	cfg.lrThld_Prevac := 5.0;	// Prevacuum pressure threshold
	// Cryo pressure threshold to start Turbo Pump before opening Valve
	cfg.lrThld_TP_SafeStartPressure := 0.01;	
	// Cryo pressure threshold to start Turbo Pump once Valve is open
	cfg.lrThld_Valve_SafeOpenPressure := 0.1;	
	cfg.tDelay := T#3S;	// Time delay before stopping Turbo Pump

	stat.bConfigured	:= TRUE;;
ELSE
	RETURN;	// Nothing to do any more
END_IF
END_METHOD

METHOD M_ExecuteControllers
VAR_INPUT
END_VAR
//
// Specific Cryo Lab Evacuation System HW configuration.
//

// Roughing Pump	
rp(	
	in_bSimulation	:= FALSE,
	in_sName		:= 'ECODRY V01',
	in_bEnable		:= ctrl.bEnable_RP,
	in_nSlaveID		:= 31,
	in_sVersion		:= 'V01',
	in_nPeriod		:= 2000);

// Turbo Molecular Pump
tp(	
	in_bSimulation	:= FALSE,
	in_sName		:= 'ATH2303M',
	in_bEnable		:= ctrl.bEnable_TP,
	in_nModel		:= 2303,
	in_bAutoMonitor	:= TRUE,
	in_nPeriod		:= 2000);

// Valve
valve(
	in_bEnable		:= ctrl.bEnable_Valve,
	in_nFeedback	:= E_CRYO_BIN_ACT_FEEDBACK.ON_AND_OFF);
END_METHOD

END_FUNCTION_BLOCK

// POUs/Subsystems/Examples/Evacuation/FB_CRYO_EVAC_PDS
FUNCTION_BLOCK FB_CRYO_EVAC_PDS EXTENDS FB_CRYO_EVAC_BASE
VAR_INPUT
END_VAR
VAR_OUTPUT
END_VAR
VAR
	rp:	FB_CRYO_PUMP_MVP030;	// Roughing Pump
	tp:	FB_CRYO_PUMP_HIPACE30;	// Turbo Molecular Pump
	
END_VAR

SUPER^();

METHOD M_Configure
VAR_INPUT
END_VAR
//
// Specific PDS IR Imager configuration.
//
IF NOT stat.bConfigured	THEN
	// MANDATORY: Set References !!!
	// If not done, system will crash !!!
	rpRef	REF=rp;
	tpRef	REF=tp;
	

	// Specific instance configuration, e.g. anything different
	// from the default values given in the cfg structure of type T_CRYO_EVAC_CFG.
	cfg.nPressGaugeType1	:= E_CRYO_SENSOR_TYPE_PRESS.PKR_360;
	cfg.nPressGaugeType2	:= E_CRYO_SENSOR_TYPE_PRESS.PKR_360;

	cfg.lrThld_Prevac := 5.0;	// Prevacuum pressure threshold
	// Cryo pressure threshold to start Turbo Pump before opening Valve
	cfg.lrThld_TP_SafeStartPressure := 0.01;	
	// Cryo pressure threshold to start Turbo Pump once Valve is open
	cfg.lrThld_Valve_SafeOpenPressure := 0.1;	
	
	cfg.tDelay := T#3S;	// Time delay before stopping Turbo Pump

	stat.bConfigured	:= TRUE;;
ELSE
	RETURN;	// Nothing to do any more
END_IF
END_METHOD

METHOD M_ExecuteControllers
VAR_INPUT
END_VAR
//
// Specific PDS IR Imager HW.
//

// Roughing Pump	
rp(	
	in_bSimulation	:= FALSE,
	in_sName		:= 'MVP 030',
	in_bEnable		:= ctrl.bEnable_RP,
	in_nModel		:= 30,
	in_bAutoMonitor	:= TRUE,
	in_nPeriod		:= 3000);

// Turbo Molecular Pump
tp(	
	in_bSimulation	:= FALSE,
	in_sName		:= 'HIPACE 30',
	in_bEnable		:= ctrl.bEnable_TP,
	in_nModel		:= 30,
	in_bAutoMonitor	:= TRUE,
	in_nPeriod		:= 3000);


valve(in_bEnable	:= ctrl.bEnable_Valve);
END_METHOD

END_FUNCTION_BLOCK

// POUs/Subsystems/Examples/Evacuation/FB_SIM_MICADO_PUMPS
FUNCTION_BLOCK FB_SIM_MICADO_PUMPS
VAR_INPUT
	in_RefPVP:	REFERENCE TO FB_CRYO_PUMP_ECODRY;
	in_RefTMP:	REFERENCE TO FB_CRYO_PUMP_ATH2303M;
	in_Delay:	TIME := T#10S;
END_VAR
VAR_OUTPUT
END_VAR
VAR
	trgStart_PVP:	R_TRIG;
	trgStart_TMP:	R_TRIG;
	trgStop_PVP:	F_TRIG;
	trgStop_TMP:	F_TRIG;
	
	timer_PVP:		TON;
	timer_TMP:		TON;
	
	bON_PVP:		BOOL := FALSE;
	bON_TMP:		BOOL := FALSE;
	
	q_PVP_Running	AT %Q*:	BOOL := TRUE;	// Active low!
	q_TMP_Ready		AT %Q*:	BOOL;
	q_TMP_Speed100	AT %Q*:	BOOL;
	
	ptrTMP_Speed:	POINTER TO DINT;
END_VAR

// Assign pointer to TMP speed.
ptrTMP_Speed	:= ADR(in_RefTMP.stat.nPumpSpeed);

// Get Start signals
trgStart_PVP(CLK:=in_RefPVP.in_bEnable);
trgStart_TMP(CLK:=in_RefTMP.in_bEnable);

// Get Stop signals
trgStop_PVP(CLK:=in_RefPVP.in_bEnable);
trgStop_TMP(CLK:=in_RefTMP.in_bEnable);

// Start timer on Start/Stop events
IF trgStart_PVP.Q THEN
	bON_PVP	:= TRUE;
	timer_PVP(IN:=FALSE);
	timer_PVP(IN:=TRUE, PT:=in_Delay/2);
ELSIF trgStop_PVP.Q THEN
	bON_PVP	:= FALSE;
	timer_PVP(IN:=FALSE);
	timer_PVP(IN:=TRUE, PT:=in_Delay/2);
END_IF

IF trgStart_TMP.Q THEN
	bON_TMP	:= TRUE;
	timer_TMP(IN:=FALSE);
	timer_TMP(IN:=TRUE, PT:=in_Delay);
ELSIF trgStop_TMP.Q THEN
	bON_TMP	:= FALSE;
	timer_TMP(IN:=FALSE);
	timer_TMP(IN:=TRUE, PT:=in_Delay * 2);
END_IF

// Execute timers
timer_PVP();
timer_TMP();

// Set outputs on timer expiry
IF timer_PVP.Q THEN
	// NOTE: PVP feedback is active low.
	IF bON_PVP THEN
		q_PVP_Running	:= FALSE;
	ELSE
		q_PVP_Running	:= TRUE;
	END_IF
END_IF

IF bON_TMP  AND (NOT timer_TMP.Q AND timer_TMP.ET > T#3S) THEN
	// Starting up.
	// Set speed > 100 rpm after 3 sec.
	ptrTMP_Speed^	:= 500;
	q_TMP_Speed100	:= TRUE;
END_IF

IF NOT bON_TMP  AND (NOT timer_TMP.Q AND timer_TMP.ET > T#5S) THEN
	// Stopping the pump.
	// Not ready after 5 sec.
	// However, the pump is still spinning.
	ptrTMP_Speed^	:= 1800;
	q_TMP_Ready		:= FALSE;
END_IF

IF timer_TMP.Q THEN
	IF bON_TMP THEN
		ptrTMP_Speed^	:= 2000;
		q_TMP_Ready	:= TRUE;
	ELSE
		ptrTMP_Speed^	:= 0;
		q_TMP_Ready		:= FALSE;
		q_TMP_Speed100	:= FALSE;
	END_IF
END_IF

END_FUNCTION_BLOCK

// POUs/Subsystems/Examples/Evacuation/FB_SIM_MICADO_VALVES
FUNCTION_BLOCK FB_SIM_MICADO_VALVES
VAR_INPUT
END_VAR
VAR_OUTPUT
END_VAR
VAR
	// Output valve control signals
	i_bON_PVV1	AT %I*:	BOOL;
	i_bON_PVV2	AT %I*:	BOOL;
	i_bON_PVV3	AT %I*:	BOOL;
	i_bON_PVV4	AT %I*:	BOOL;
	i_bON_GBV	AT %I*:	BOOL;
	
	
	// Simulation of ON/open feedback signal
	q_bON_PVV1	AT %Q*:	BOOL := FALSE;
	q_bON_PVV2	AT %Q*:	BOOL := FALSE;
	q_bON_PVV3	AT %Q*:	BOOL := FALSE;
	q_bON_PVV4	AT %Q*:	BOOL := FALSE;
	q_bON_GBV	AT %Q*:	BOOL := FALSE;
	
	// Simulation of OFF/closed feedback signal
	q_bOFF_PVV1	AT %Q*:	BOOL := TRUE;
	q_bOFF_PVV2	AT %Q*:	BOOL := TRUE;
	q_bOFF_PVV3	AT %Q*:	BOOL := TRUE;
	q_bOFF_PVV4	AT %Q*:	BOOL := TRUE;
	q_bOFF_GBV	AT %Q*:	BOOL := TRUE;
	

END_VAR

// ON signals are active low
q_bON_PVV1	:= i_bON_PVV1;
q_bON_PVV2	:= i_bON_PVV2;
q_bON_PVV3	:= i_bON_PVV3;
q_bON_PVV4	:= i_bON_PVV4;
q_bON_GBV	:= i_bON_GBV;


// OFF signals are active low
q_bOFF_PVV1	:= NOT i_bON_PVV1;
q_bOFF_PVV2	:= NOT i_bON_PVV2;
q_bOFF_PVV3	:= NOT i_bON_PVV3;
q_bOFF_PVV4	:= NOT i_bON_PVV4;
q_bOFF_GBV	:= NOT i_bON_GBV;

END_FUNCTION_BLOCK

// POUs/Subsystems/Examples/LN2_Precooling/FB_CRYO_LN2_PRECOOL
FUNCTION_BLOCK FB_CRYO_LN2_PRECOOL EXTENDS FB_CRYO_GEN_CTRL_BASE
VAR_INPUT
	in_lrTempK:				LREAL;			// Temperature input value [K]
	in_bTempValid:			BOOL := TRUE;	// Temperature Valid flag
	// Two parameters for decision making
	in_lrTempValveOpen:		LREAL := 91.27;		// Open  valve if temperature above this value [K]
	in_lrTempValveClose:	LREAL := 79.148;	// Close valve if temperature below this value [K]
END_VAR
VAR_OUTPUT
END_VAR
VAR
	// Status structure
	{attribute 'OPC.UA.DA' := '1'}
	stat:				T_CRYO_GEN_CTRL_STATUS_BASE;
	
	// LN2 valve
	valve:				FB_CRYO_VALVE_CTRL;
	bEnable_valve:		BOOL := FALSE;	// Valve open when bEnable_valve = TRUE
		

END_VAR

SUPER^();

METHOD M_ActionOffExecute
VAR_INPUT
END_VAR
//
// In this method the Enable flag of the valve is set to FALSE,
// meaning close the valve.
// 
// In the corresponding Activity M_ActivitySwitchingOff(), 
// the completion of the CLOSE/OFF command will be checked.
//
timer(IN:=FALSE);	// Reset Timer - mandatory!

// Close the valve
bEnable_valve	:= FALSE;
END_METHOD

METHOD M_ActionOnExecute
VAR_INPUT
END_VAR
//
// In this method the Enable flag of the valve is set to TRUE,
// meaning open the valve.
// 
// In the corresponding Activity M_ActivitySwitchingOn(), 
// the completion of the OPEN/ON command will be checked.
//
timer(IN:=FALSE);	// Reset Timer - mandatory!

// Close the valve
bEnable_valve	:= TRUE;
END_METHOD

METHOD M_ActivitySwitchingOff : BOOL
VAR_INPUT
END_VAR
//
// Wait for the valve to CLOSE/OFF.
// The valve state is available in its status structure.
// When complete, the method shall return TRUE, otherwise FALSE.


//
// Execute the timer - mandatory.
// Timer expiry is checked in M_ProcessEvents().
//
timer(IN:=TRUE, PT:=UDINT_TO_TIME(in_nTimeout));
	
// If valve is closed, return TRUE, otherwise FALSE.
IF valve.stat.bActOFF THEN
	M_ActivitySwitchingOff := TRUE;
ELSE
	M_ActivitySwitchingOff := FALSE;
END_IF
END_METHOD

METHOD M_ActivitySwitchingOn : BOOL
VAR_INPUT
END_VAR
//
// Wait for the valve to OPEN/ON.
// The valve state is available in its status structure.
// When complete, the method shall return TRUE, otherwise FALSE.


//
// Execute the timer - mandatory.
// Timer expiry is checked in M_ProcessEvents().
//
timer(IN:=TRUE, PT:=UDINT_TO_TIME(in_nTimeout));
	
// If valve is open, return TRUE, otherwise FALSE.
IF valve.stat.bActON THEN
	M_ActivitySwitchingOn := TRUE;
ELSE
	M_ActivitySwitchingOn := FALSE;
END_IF
END_METHOD

METHOD M_Configure
VAR_INPUT
END_VAR
// Configure the system and set the bConfigured flag to TRUE.

(*
	TODO USER: 
	- Set references to extended structures. e.g.
	     statRef REF=stat;
	- Configure the system.
*)

//	MUST be the very first line!!!
statRef REF=stat;

// The system has been configured
bConfigured := TRUE;
END_METHOD

METHOD M_ControlLoop : BOOL
VAR_INPUT
END_VAR
//
// This method implements the logic for controlling the LN2 valve.
// 
// The return value indicates if the valve should be OPEN/TRUE or CLOSED/FALSE
//
	
CASE statRef.nState OF
	E_CRYO_BIN_CTRL_STATE.ACTIVE_SWITCHING_ON,
	E_CRYO_BIN_CTRL_STATE.ACTIVE_ON:
		IF in_bTempValid AND in_lrTempK < in_lrTempValveClose THEN
			// Temperature too low.
			// Close the valve to stop cooling.
			M_ControlLoop	:= FALSE;
		ELSE
			// Keep the valve open
			M_ControlLoop	:= TRUE;
		END_IF

	E_CRYO_BIN_CTRL_STATE.ACTIVE_SWITCHING_OFF,
	E_CRYO_BIN_CTRL_STATE.ACTIVE_OFF:
		IF in_bTempValid AND in_lrTempK > in_lrTempValveOpen THEN
			// Temperature too high.
			// Open the valve to start cooling.
			M_ControlLoop	:= TRUE;
		ELSE
			// Keep the valve closed
			M_ControlLoop	:= FALSE;
		END_IF
ELSE
	// Keep the valve closed
	M_ControlLoop	:= FALSE;
END_CASE
END_METHOD

METHOD M_ExecuteActuators
VAR_INPUT
END_VAR
(*
	TODO USER: Execute all actuators, e.g. valve, heater, etc.
*)

valve(	in_nTimeout	:= 3000, 
		in_bEnable	:= bEnable_valve);
END_METHOD

METHOD M_IsError : BOOL
VAR_INPUT
END_VAR
//
// Check all possible failure conditions.
//
// This includes:
// - Configuration,
// - Validity of temperature reading,
// - Valve failure.
// 
// Return TRUE in case of errors.
// Set error description as well.
//
IF in_lrTempValveClose >= in_lrTempValveOpen THEN
	// The temperatue at which valve opens must be
	// higher than the one at which it closes.
	M_IsError	:= TRUE;
	stat.sError	:= 'ERROR: Wrong temperature limits!';
ELSIF NOT in_bTempValid	THEN
	// Temperature reading invalid.
	M_IsError	:= TRUE;
	stat.sError	:= 'ERROR: Reference temperature invalid!';
ELSIF valve.stat.bError 	THEN
	// Valve has failed.
	M_IsError	:= TRUE;
	stat.sError	:= 'ERROR: Valve failure!';
ELSE
	M_IsError	:= FALSE;
END_IF
END_METHOD

METHOD M_SetStatus
VAR_INPUT
END_VAR
// Execute M_SetStatus() of the base FB
SUPER^.M_SetStatus();


// Correct for LN2 specific labels

CASE statRef.nState OF
	
	E_CRYO_BIN_CTRL_STATE.ACTIVE_OFF:
	statRef.sState	:= 'ACTIVE_VALVE_CLOSED';
	
	E_CRYO_BIN_CTRL_STATE.ACTIVE_ON:
	statRef.sState	:= 'ACTIVE_VALVE_OPEN';
	
	E_CRYO_BIN_CTRL_STATE.ACTIVE_SWITCHING_ON:
	statRef.sState	:= 'OPENING VALVE...';
	
	E_CRYO_BIN_CTRL_STATE.ACTIVE_SWITCHING_OFF:
	statRef.sState	:= 'CLOSING VALVE...';
	
END_CASE
END_METHOD

END_FUNCTION_BLOCK

// POUs/Subsystems/Examples/LN2_Precooling/FB_SIM_LN2_PRECOOL
FUNCTION_BLOCK FB_SIM_LN2_PRECOOL
VAR_INPUT
	ln2Ref:	REFERENCE TO FB_CRYO_LN2_PRECOOL;
END_VAR
VAR_OUTPUT
	lrTempK:	LREAL;	// Simulated temperature value [K]
END_VAR
VAR
	SIM_ln2_temp:	FB_CRYO_SIM_TEMPERATURE;	// Simulated temperature FB
	
	trgEnable:		R_TRIG;						// Precooling  enable change trigger
	trgDisable:		F_TRIG;						// Precooling disable change trigger
	trgState:		R_TRIG;						// State change trigger

	nState:			E_CRYO_BIN_CTRL_STATE	:= E_CRYO_BIN_CTRL_STATE.NONE;
	
END_VAR

// Detect change of LN2 system Enable 
trgEnable(CLK := ln2Ref.in_bEnable);

// Detect change of LN2 system Disable 
trgDisable(CLK := ln2Ref.in_bEnable);

// Detect change of LN2 system State 
trgState(CLK := (	(ln2Ref.stat.nState = E_CRYO_BIN_CTRL_STATE.ACTIVE_ON OR 
					 ln2Ref.stat.nState = E_CRYO_BIN_CTRL_STATE.ACTIVE_OFF) 	AND 
					ln2Ref.stat.nState <> nState));

IF trgEnable.Q	THEN
	// System enabled.

	// Save current state
	nState	:= ln2Ref.stat.nState;
	
	// Start changing temperature just to get the system 
	// working for the first time.
	IF SIM_ln2_temp.lrTempK >= ln2Ref.in_lrTempValveClose	THEN
		// Lower simulated temperature to lower limit -1 deg in 5 sec.
		SIM_ln2_temp.M_RampTo(ln2Ref.in_lrTempValveClose - 1, 5000);
	ELSE
		// Rise simulated temperature to upper limit +1 deg in 5 sec.
		SIM_ln2_temp.M_RampTo(ln2Ref.in_lrTempValveOpen + 1, 5000);
	END_IF
ELSIF trgDisable.Q	THEN
	// System disabled. Stop the temperature ramp.
	SIM_ln2_temp.M_Stop();	
ELSIF ln2Ref.in_bEnable AND trgState.Q	THEN
	// State of enabled system changed.
	// Save new state
	nState	:= ln2Ref.stat.nState;
	
	// Start a ramp, depending on the new state.
	IF ln2Ref.stat.nState = E_CRYO_BIN_CTRL_STATE.ACTIVE_ON	THEN
		// Valve open, the temperature should start falling.
		// Ramp it down to the CLOSE limit minus 1 deg in 10 sec.
		SIM_ln2_temp.M_RampTo(ln2Ref.in_lrTempValveClose - 1.0, 10000);
	ELSIF ln2Ref.stat.nState = E_CRYO_BIN_CTRL_STATE.ACTIVE_OFF	THEN
		// Valve closed, the temperature should start rising.
		// Ramp it up to the OPEN limit plus 1 deg in 10 sec.
		SIM_ln2_temp.M_RampTo(ln2Ref.in_lrTempValveOpen + 1.0, 10000);
	END_IF
END_IF


// Execute temperature simulator FB.
SIM_ln2_temp();

// Assign the simulated temperature to the output var
lrTempK	:= SIM_ln2_temp.lrTempK;

END_FUNCTION_BLOCK

// POUs/Utilities/FB_CRYO_THLD_BASE
FUNCTION_BLOCK FB_CRYO_THLD_BASE
VAR_INPUT
	in_nMode:		E_CRYO_THLD_MODE := E_CRYO_THLD_MODE.FIXED;
	in_aThld:		ARRAY [1..4] OF LREAL;	// Array of fixed thresholds. See E_CRYO_ALARM_LEVELS and E_CRYO_ALARM_IDX.
	in_aThldDelay:	ARRAY [1..4] OF UDINT;	// Array of delays for each threshold [ms].
	in_lrHyst:		LREAL := 0.0;			// Hysteresis value, percent or absolute (see in_bHystPct)
	in_bHystPct:	BOOL := TRUE;			// If TRUE, hysteresis is in %, otherwise absolute value.
	in_lrValue:		LREAL;					// Value to compare against the thresholds
	in_lrPar1:		LREAL := 0.0;			// Par1, e.g. temperature, for ACTIVE thresholds
END_VAR
VAR_OUTPUT
	out_aThld:			ARRAY [1..4] OF LREAL;	// Active thresholds
	out_nAlarmState:	E_CRYO_ALARM_LEVEL	:= E_CRYO_ALARM_LEVEL.NORMAL;	// Alarm state, e.g. ALARM_HIGH
	out_sAlarmState:	STRING := 'NORMAL';	// Alarm state as a string, e.g. 'ALARM HIGH'
END_VAR
VAR
	timer:	TON;
END_VAR

// Set thresholds
M_SetThresholds();

// Compare input value against the thresholds
M_CheckAlarms();

METHOD M_CheckAlarms : BOOL
VAR_INPUT
END_VAR
VAR
	lrHyst:	LREAL;
END_VAR

// Execute the delay timer.
timer();

//
// Check the input value against the thresholds
// and set alarms and warnings.
// If configured for, activate alarms after a delay.
// Note: the value is compared against the OUT Thresholds !!!
//
CASE out_nAlarmState OF
	E_CRYO_ALARM_LEVEL.NORMAL:
		IF in_lrValue > out_aThld[E_CRYO_ALARM_IDX.ALARM_HIGH] THEN
			IF in_aThldDelay[E_CRYO_ALARM_IDX.ALARM_HIGH] > 0	THEN
				// Activation delay is configured.
				// Start the timer and change state to WARNING_HIGH.
				timer(IN:=FALSE);
				timer(IN:=TRUE, PT:=UDINT_TO_TIME(in_aThldDelay[E_CRYO_ALARM_IDX.ALARM_HIGH]));
				out_nAlarmState	:= E_CRYO_ALARM_LEVEL.WARNING_HIGH;
			ELSE
				timer(IN:=FALSE);
				out_nAlarmState	:= E_CRYO_ALARM_LEVEL.ALARM_HIGH;
			END_IF
		ELSIF in_lrValue < out_aThld[E_CRYO_ALARM_IDX.ALARM_LOW] THEN
			IF in_aThldDelay[E_CRYO_ALARM_IDX.ALARM_LOW] > 0	THEN
				// Activation delay is configured.
				// Start the timer and change state to WARNING_LOW.
				timer(IN:=FALSE);
				timer(IN:=TRUE, PT:=UDINT_TO_TIME(in_aThldDelay[E_CRYO_ALARM_IDX.ALARM_LOW]));
				out_nAlarmState	:= E_CRYO_ALARM_LEVEL.WARNING_LOW;
			ELSE
				timer(IN:=FALSE);
				out_nAlarmState	:= E_CRYO_ALARM_LEVEL.ALARM_LOW;
			END_IF
		ELSIF in_lrValue > out_aThld[E_CRYO_ALARM_IDX.WARNING_HIGH] THEN
			IF in_aThldDelay[E_CRYO_ALARM_IDX.WARNING_HIGH] > 0	THEN
				// Activation delay is configured.
				// Activate the warning once the timer expires.
				timer(IN:=TRUE, PT:=UDINT_TO_TIME(in_aThldDelay[E_CRYO_ALARM_IDX.WARNING_HIGH]));
				IF timer.Q	THEN
					IF in_lrValue > out_aThld[E_CRYO_ALARM_IDX.ALARM_HIGH] THEN
						// It might be that due to the delay the alarm level has been reached.
						out_nAlarmState	:= E_CRYO_ALARM_LEVEL.ALARM_HIGH;
					ELSE
						out_nAlarmState	:= E_CRYO_ALARM_LEVEL.WARNING_HIGH;
					END_IF
				END_IF
			ELSE
				timer(IN:=FALSE);
				out_nAlarmState	:= E_CRYO_ALARM_LEVEL.WARNING_HIGH;
			END_IF
		ELSIF	in_lrValue < out_aThld[E_CRYO_ALARM_IDX.WARNING_LOW]	THEN
			IF in_aThldDelay[E_CRYO_ALARM_IDX.WARNING_LOW] > 0	THEN
				// Activation delay is configured.
				// Activate the warning once the timer expires.
				timer(IN:=TRUE, PT:=UDINT_TO_TIME(in_aThldDelay[E_CRYO_ALARM_IDX.WARNING_LOW]));
				IF timer.Q	THEN
					IF in_lrValue < out_aThld[E_CRYO_ALARM_IDX.ALARM_LOW] THEN
						// It might be that due to the delay the alarm level has been reached.
						out_nAlarmState	:= E_CRYO_ALARM_LEVEL.ALARM_LOW;
					ELSE
						out_nAlarmState	:= E_CRYO_ALARM_LEVEL.WARNING_LOW;
					END_IF
				END_IF
			ELSE
				timer(IN:=FALSE);
				out_nAlarmState	:= E_CRYO_ALARM_LEVEL.WARNING_LOW;
			END_IF
		ELSE
			timer(IN:=FALSE);
		END_IF
	E_CRYO_ALARM_LEVEL.WARNING_HIGH:
		lrHyst	:= M_GetHysteresis(E_CRYO_ALARM_IDX.WARNING_HIGH);
		IF	in_lrValue > out_aThld[E_CRYO_ALARM_IDX.ALARM_HIGH]	THEN
			IF in_aThldDelay[E_CRYO_ALARM_IDX.ALARM_HIGH] > 0	THEN
				// Activation delay is configured.
				// Activate the alarm once the timer expires.
				timer(IN:=TRUE, PT:=UDINT_TO_TIME(in_aThldDelay[E_CRYO_ALARM_IDX.ALARM_HIGH]));
				IF timer.Q	THEN
					out_nAlarmState	:= E_CRYO_ALARM_LEVEL.ALARM_HIGH;
				END_IF
			ELSE
				timer(IN:=FALSE);
				out_nAlarmState	:= E_CRYO_ALARM_LEVEL.ALARM_HIGH;
			END_IF
		ELSIF in_lrValue < (out_aThld[E_CRYO_ALARM_IDX.WARNING_HIGH] - lrHyst) THEN
			timer(IN:=FALSE);
			out_nAlarmState	:= E_CRYO_ALARM_LEVEL.NORMAL;
		ELSE
			timer(IN:=FALSE);
		END_IF
	E_CRYO_ALARM_LEVEL.WARNING_LOW:
		lrHyst	:= M_GetHysteresis(E_CRYO_ALARM_IDX.WARNING_LOW);
		IF	in_lrValue < out_aThld[E_CRYO_ALARM_IDX.ALARM_LOW]	THEN
			IF in_aThldDelay[E_CRYO_ALARM_IDX.ALARM_LOW] > 0	THEN
				// Activation delay is configured.
				// Activate the alarm once the timer expires.
				timer(IN:=TRUE, PT:=UDINT_TO_TIME(in_aThldDelay[E_CRYO_ALARM_IDX.ALARM_LOW]));
				IF timer.Q	THEN
					out_nAlarmState	:= E_CRYO_ALARM_LEVEL.ALARM_LOW;
				END_IF
			ELSE
				timer(IN:=FALSE);
				out_nAlarmState	:= E_CRYO_ALARM_LEVEL.ALARM_LOW;
			END_IF
		ELSIF in_lrValue > (out_aThld[E_CRYO_ALARM_IDX.WARNING_LOW] + lrHyst) THEN
			timer(IN:=FALSE);
			out_nAlarmState	:= E_CRYO_ALARM_LEVEL.NORMAL;
		ELSE
			timer(IN:=FALSE);
		END_IF
	E_CRYO_ALARM_LEVEL.ALARM_HIGH:
		lrHyst	:= M_GetHysteresis(E_CRYO_ALARM_IDX.ALARM_HIGH);
		IF in_lrValue < (out_aThld[E_CRYO_ALARM_IDX.ALARM_HIGH] - lrHyst) THEN
			out_nAlarmState	:= E_CRYO_ALARM_LEVEL.WARNING_HIGH;
		END_IF
	E_CRYO_ALARM_LEVEL.ALARM_LOW:
		lrHyst	:= M_GetHysteresis(E_CRYO_ALARM_IDX.ALARM_LOW);
		IF in_lrValue > (out_aThld[E_CRYO_ALARM_IDX.ALARM_LOW] + lrHyst) THEN
			out_nAlarmState	:= E_CRYO_ALARM_LEVEL.WARNING_LOW;
		END_IF
END_CASE

// Set alarm level labels
M_UserSetLabel(out_nAlarmState);
END_METHOD

METHOD M_GetHysteresis : LREAL
VAR_INPUT
	in_nIndex:	E_CRYO_ALARM_IDX;
END_VAR
VAR
	lrHyst:	LREAL;
END_VAR
//
// Get the absolute value of hysteresis.
// 
IF in_bHystPct THEN
	// The vaue is given as percentage of threshold.
	lrHyst	:= in_aThld[in_nIndex] * in_lrHyst / 100.0;
ELSE
	// The vaue is given as absolute value.
	lrHyst	:= in_lrHyst;
END_IF

M_GetHysteresis	:= ABS(lrHyst);
END_METHOD

METHOD M_SetThresholds : BOOL
VAR_INPUT
END_VAR
VAR
	i:	INT;
END_VAR
CASE in_nMode OF
	E_CRYO_THLD_MODE.FIXED:
		// Take the input array for thresholds
		FOR i:=1 TO 4 DO
			out_aThld[i]	:= in_aThld[i];
		END_FOR
	E_CRYO_THLD_MODE.ACTIVE:
		// Dynamically set thresholds
		M_UserSetActiveThresholds();
	E_CRYO_THLD_MODE.LAST_ACTIVE:
		// Keep last thresholds. Don't do anything.
		;
END_CASE
END_METHOD

METHOD M_UserSetActiveThresholds : BOOL
// This is a Dummy implementation of active thresholds.
// TODO User: Define specific implementation.
VAR_INPUT
END_VAR
VAR
	i:	INT;
END_VAR
// TODO User
// Define specific implementation.
// This is just an example.
//
out_aThld[E_CRYO_ALARM_IDX.ALARM_LOW]	:= in_aThld[E_CRYO_ALARM_IDX.ALARM_LOW]    + in_lrPar1;
out_aThld[E_CRYO_ALARM_IDX.WARNING_LOW]	:= in_aThld[E_CRYO_ALARM_IDX.WARNING_LOW]  + in_lrPar1;
out_aThld[E_CRYO_ALARM_IDX.WARNING_HIGH]	:= in_aThld[E_CRYO_ALARM_IDX.WARNING_HIGH] - in_lrPar1;
out_aThld[E_CRYO_ALARM_IDX.ALARM_HIGH]	:= in_aThld[E_CRYO_ALARM_IDX.ALARM_HIGH]   - in_lrPar1;
END_METHOD

METHOD M_UserSetLabel : BOOL
VAR_INPUT
	in_nLevel:	E_CRYO_ALARM_LEVEL;
END_VAR
//
// Set labels depending on the alarm level.
// This is the default implementation.
// To be overwritten by User if different labels are needed.
//
CASE in_nLevel OF
	E_CRYO_ALARM_LEVEL.ALARM_LOW:
		out_sAlarmState	:= 'ALARM LOW';
	E_CRYO_ALARM_LEVEL.WARNING_LOW:
		out_sAlarmState	:= 'WARNING LOW';
	E_CRYO_ALARM_LEVEL.NORMAL:
		out_sAlarmState	:= 'NORMAL';
	E_CRYO_ALARM_LEVEL.WARNING_HIGH:
		out_sAlarmState	:= 'WARNING HIGH';
	E_CRYO_ALARM_LEVEL.ALARM_HIGH:
		out_sAlarmState	:= 'ALARM HIGH';
END_CASE
END_METHOD

END_FUNCTION_BLOCK

// POUs/MAIN
PROGRAM MAIN
VAR
	
	
	{attribute 'OPC.UA.DA' := '1'}
	Cryo_Ctrl:	FB_CRYO_CTRL;
	
	
	{attribute 'OPC.UA.DA' := '1'}
	SIM_Cryo_Ctrl:	FB_CRYO_SIM_CTRL;
	
	//
	// Pressure voting system testing
	//
	P1_1:	FB_CRYO_SENSOR_PRESSURE;
	P1_2:	FB_CRYO_SENSOR_PRESSURE;
	P1_3:	FB_CRYO_SENSOR_PRESSURE;
	P1_4:	FB_CRYO_SENSOR_PRESSURE;
	P1_5:	FB_CRYO_SENSOR_PRESSURE;
	P1:		FB_CRYO_PRESSURE_VOTE;	// Voting of P1_1..P1_5

	nVoteMethod:		E_CRYO_VOTE	:=E_CRYO_VOTE.V_3oo5;
	bP1_Sim:			BOOL := FALSE;
	SIM_Pressure_P1:	FB_CRYO_SIM_PRESSURE;		// P1 Pressure simulator
	pressOR_P1:			FB_CRYO_CMD_OVERRIDE;

	////////////////////////////
	// Temperature testing
	//
	T1:		FB_CRYO_SENSOR_TEMPERATURE;
	T2:		FB_CRYO_TEMPERATURE;
	nRampPeriodSec:		UDINT := 60;	// Ramp measurement period [sec]. Default 60 sec.
	tempOR_T2:	FB_CRYO_CMD_OVERRIDE;
	simT2:		BOOL;
	////////////////////////////
	
	
	//////////////////////////////////////////////////////////////////
	
	//
	// Threshold testing
	//
	thld1:		FB_CRYO_THLD_BASE;	// Threshold handling
	
	// Threshold levels in format
	// [<alarm low>, <warning low>, <warning high>, <alarm high>]
	aThlds:		ARRAY [1..4] OF LREAL	:= [-80.0, -60.0, 40.0, 80.0];
	aThldDelay:	ARRAY [1..4] OF UDINT	:= [1000, 0, 2000, 0];
	nThldMode:	E_CRYO_THLD_MODE := E_CRYO_THLD_MODE.FIXED;	// Threshold check mode
	lrHyst:		LREAL	:= 10.0;	// Threshold hysteresis
	lrThldRef:	LREAL	:= 0.0;		// Threshold reference for User defined active thresholds
	
	SIM_thld1:	FB_CRYO_SIM_SINE;	// Simulated signal for threshold testing
	SIM_thld2:	FB_CRYO_SIM_SINE;	// Simulated signal for threshold testing
	nSimPer1:	UDINT := 60000;		// Period [ms] of simulated sine curve #1
	nSimPer2:	UDINT := 16000;		// Period [ms] of simulated sine curve #2
	
	/////////////////////////////////////////////////////////////////////////
	/////////////////////////////////////////////////////////////////////////

	///////////////////
	// Lakeshore 336
	///////////////////
	// Lakeshore 336 (Ethernet interface)
	{attribute 'OPC.UA.DA' := '1'}
	LS336_TCP:		FB_LAKESHORE_TCP;		// LakeShore based on FB_TCP_CLIENT



///////////////////////////////////////////////////////////////////
// Pumps and evacuations
///////////////////////////////////////////////////////////////////
	
	evac_pds:	FB_CRYO_EVAC_PDS;

	evac_lab:	FB_CRYO_EVAC_ECODRY_ATH2303M;	
	
	evac_micado:	FB_CRYO_EVAC_MICADO;

	// Cryostat pressure (sensor and evaluation)
	cryo_lab_press1:	FB_CRYO_SENSOR_PRESSURE;	// Cryostat pressure gauge #1
	cryo_lab_pressure:	FB_CRYO_PRESSURE_VOTE;		// Cryostat pressure 
	
	// Flags to control start/stop of pumps
	bEnable_evac_pds:	BOOL;
	bEnable_evac_lab:	BOOL;
	bEnable_evac_mic:	BOOL;
	
	// Simulation flags
	bSim_cryo_lab_pressure:	BOOL;
	
	
	//////////////////////////////
	// SUNPOWER Cryotel GT Cooler
	//////////////////////////////
	cooler:			FB_CRYO_CRYOTELGT;
	bEnable_cooler:	BOOL;
	
	
	///////////////////
	// MICADO
	///////////////////
	sensor_VAGF1:	FB_CRYO_SENSOR_PRESSURE;	// Cryo pressure gauge VAG F1
	sensor_VAGF2:	FB_CRYO_SENSOR_PRESSURE;	// Cryo pressure gauge VAG F2
	sensor_VAGG1:	FB_CRYO_SENSOR_PRESSURE;	// Cryo pressure gauge VAG G1
	sensor_VAGG2:	FB_CRYO_SENSOR_PRESSURE;	// Cryo pressure gauge VAG G2
	VAGF:	FB_CRYO_PRESSURE_VOTE;				// Cryo pressure F
	VAGG:	FB_CRYO_PRESSURE_VOTE;				// Cryo pressure G

	// Valve Command handling
	cmdPVV1:	FB_CRYO_ACTUATOR_CMD;
	bCmdPVV1:	BOOL;	// Open/Close command for PVV1
	bIntlkPVV1:	BOOL;	// Interlock for PVV1
	
	///////////////////
	// Simulation
	/////////////////
	
	mic_valves:	FB_SIM_MICADO_VALVES;
	mic_pumps:	FB_SIM_MICADO_PUMPS;
	
	// Pressure values
	q_nVAG1		AT %Q*:	INT := 30000;
	q_nVAG2		AT %Q*:	INT := 30000;
	q_nVAG3		AT %Q*:	INT := 30000;
	q_nVAGF1	AT %Q*:	INT := 30000;
	q_nVAGF2	AT %Q*:	INT := 30000;
	q_nVAGG1	AT %Q*:	INT := 30000;
	q_nVAGG2	AT %Q*:	INT := 30000;
	
	// Used for simulated toggle signal
	pSim:	FB_CRYO_SIM_PRESSURE;
	
	q_nCouplerState	AT %Q*:	INT := 8;
	
	///////////////////////
	// Pressure Ramp Test
	///////////////////////
	SIM_P1:		FB_CRYO_SIM_PRESSURE;
	bStartRamp:	BOOL;
	
	// Actuator test
	actuator:	FB_CRYO_BIN_ACT;
	
	// FB_CRYO_ACTUATOR_CMD test
	Valve1:		FB_CRYO_VALVE_CTRL;		// No override possible
	Valve2:		FB_CRYO_VALVE_CTRL;		// Override possible
	cmdValve2:	FB_CRYO_ACTUATOR_CMD;	// Handling of Valve2 command
	// System commands for Valve1 and Valve2
	bEnable_Valve1:	BOOL;
	bEnable_Valve2:	BOOL;
	
	// FB_CRYO_CMD_OVERRIDE test
	cmdOverrideTest:	FB_CRYO_CMD_OVERRIDE;
	bEnable_OverrideTest:	BOOL;

	//////////////////////////////
	// Testing FB_CRYO_LN2_PRECOOL
	//////////////////////////////
	ln2_ctrl:			FB_CRYO_LN2_PRECOOL;	// LN2 controller
	SIM_ln2:			FB_SIM_LN2_PRECOOL;		// LN2 temperature simulator
	bEnable_ln2_ctrl:	BOOL;					// Flag to activate/deactivate LN2 controller
	
	/////////////////////////////////////////////
	// Testing IO-Link FB_CRYO_SBG232 Flowmeter
	/////////////////////////////////////////////
	
	sbg232:		FB_CRYO_SBG232;
	sbg232_sim:	FB_CRYO_SBG232;
	
	SIM_sbg232:	FB_CRYO_SIM_SBG232;
	
END_VAR

	
Cryo_Ctrl();

SIM_Cryo_Ctrl(in_ptr_Cryo_Ctrl:=ADR(Cryo_Ctrl));


//
// Pressure voting system testing
//
SIM_Pressure_P1(in_nType:=E_CRYO_SENSOR_TYPE_PRESS.PKR_360);


// Measuring point P1 - five sensors
P1_1(in_nType:=E_CRYO_SENSOR_TYPE_PRESS.PKR_360, in_nSampleTime:=100);
P1_2(in_nType:=E_CRYO_SENSOR_TYPE_PRESS.PKR_360, in_nSampleTime:=100);
P1_3(in_nType:=E_CRYO_SENSOR_TYPE_PRESS.PKR_360, in_nSampleTime:=100);
P1_4(in_nType:=E_CRYO_SENSOR_TYPE_PRESS.PKR_360, in_nSampleTime:=100);
P1_5(in_nType:=E_CRYO_SENSOR_TYPE_PRESS.PKR_360, in_nSampleTime:=100);

pressOR_P1(in_bEnable:=bP1_Sim);	// Override of simulation flag
P1(	in_bSimulation	:= pressOR_P1.out_bEnable,
	in_nNumSensor	:= 5, 
	in_nVoteMethod	:= nVoteMethod,
	in_pSensor1		:= ADR(P1_1),
	in_pSensor2		:= ADR(P1_2),
	in_pSensor3		:= ADR(P1_3),
	in_pSensor4		:= ADR(P1_4),
	in_pSensor5		:= ADR(P1_5));

	
//
// Temperature testing
//
T1(in_nRampPeriodSec:=nRampPeriodSec);
tempOR_T2(in_bEnable:=simT2);
T2(in_bSimulation:=tempOR_T2.out_bEnable);


//
// Threshold testing
//
// Simulated sensor value is the combination of two 
// sine wave curves with different period and amplitude.
SIM_thld1(in_lrAmplitude := 95.0, in_nPeriod := nSimPer1);
SIM_thld2(in_lrAmplitude := 20.0, in_nPeriod := nSimPer2);

// Threshold instance
// in_lrValue is the sum of two curves.
thld1(
	in_nMode		:= nThldMode,
	in_aThld		:= aThlds,
	in_aThldDelay	:= aThldDelay,
	in_lrHyst 		:= lrHyst,
	in_lrValue 		:= SIM_thld1.out_lrValue + SIM_thld2.out_lrValue,
	in_lrPar1		:= lrThldRef);


///////////////////
// Lakeshore 336
///////////////////
LS336_TCP(	in_sName			:= 'LS336_TCP',		// Device name
			in_bSimulation		:= FALSE,			// Device simulation
			in_bAutoMonitor		:= TRUE,			// Go to OPERATIONAL, a MUST!
			in_nModel			:= 336,				// Model number
			in_nPeriod			:= 1000,			// Update period [ms]
			in_sCmdSuffix		:= '$0A',			// Command suffix LF
			in_sReplySuffix		:= '$0A',			// Reply suffix LF
			in_sDeviceTcpIpAdr	:= '192.168.0.80', 	// Lakeshore IP address
			in_nDeviceTcpPort	:= 7777);			// Lakeshore port

(*
// Configure Lakeshore for Warmup.
// To be executed only once at the start of the warmup.
LS336_TCP.M_RampEnable(
	in_nPID_A_P			:= 10, 
	in_nPID_A_I			:= 50, 
	in_nPID_A_D			:= 20, 
	in_nHeater_Range	:= 4, 
	in_lrCtrlRamp		:= 1.0, 	// 1.0 deg/min
	in_lrSetpoint_A		:= 293.15);	// 20 deg Celsius
*)			
	
	
///////////////////////////////////////////////////////////////////
// Pumps code
///////////////////////////////////////////////////////////////////
// Handle ELT Cryo Lab Cryostat pressure
cryo_lab_press1(in_nType := E_CRYO_SENSOR_TYPE_PRESS.PKR_250, in_nSampleTime := 100);
cryo_lab_pressure(
	in_bSimulation	:= bSim_cryo_lab_pressure,
	in_nNumSensor	:= 2,	// In reality, there is only one pressure sensor connected
	in_nVoteMethod	:= E_CRYO_VOTE.V_1oo2,
	in_pSensor1		:= ADR(cryo_lab_press1));



// Evacuation system for the PDS IR Imager
evac_pds(in_bEnable	:= bEnable_evac_pds);

// Evacuation system in the ELT Cryo Lab
evac_lab(
	in_bEnable			:= bEnable_evac_lab, 
	in_lrCryoPressure	:= cryo_lab_pressure.stat.lrPressure);


//////////////////////////////
// SUNPOWER Cryotel GT Cooler
//////////////////////////////
cooler(	in_sName		:= 'CryotelGT',
		in_bSimulation	:= TRUE,
		in_bAutoMonitor	:= TRUE,
		in_bEnable		:= bEnable_cooler);

	
	
///////////////
// MICADO
///////////////

pSim();	// Just to have a simulated Toggle signal.

// Simulation of MICADO valves
mic_valves();	

// Simulation of MICADO pumps
mic_pumps(in_RefPVP:=evac_micado.rp, in_RefTMP:=evac_micado.tp);	



// MICADO Cryostat pressures
sensor_VAGF1(in_nType := E_CRYO_SENSOR_TYPE_PRESS.PKR_360,	in_nSampleTime := 100);
sensor_VAGF2(in_nType := E_CRYO_SENSOR_TYPE_PRESS.PKR_360,	in_nSampleTime := 100);
sensor_VAGG1(in_nType := E_CRYO_SENSOR_TYPE_PRESS.PKR_360,	in_nSampleTime := 100);
sensor_VAGG2(in_nType := E_CRYO_SENSOR_TYPE_PRESS.PKR_360,	in_nSampleTime := 100);

VAGF(
	in_bSimulation	:= FALSE,
	in_nNumSensor	:= 2,
	in_nVoteMethod	:= E_CRYO_VOTE.V_1oo2,
	in_pSensor1		:= ADR(sensor_VAGF1),
	in_pSensor2		:= ADR(sensor_VAGF2));

VAGG(
	in_bSimulation	:= FALSE,
	in_nNumSensor	:= 2,
	in_nVoteMethod	:= E_CRYO_VOTE.V_1oo2,
	in_pSensor1		:= ADR(sensor_VAGG1),
	in_pSensor2		:= ADR(sensor_VAGG2));

	
// MICADO evacuation system
cmdPVV1(in_bEnable:=bCmdPVV1,in_bInterlock:=bIntlkPVV1);	// Handling of PVV1 commands

evac_micado(
	in_bEnable		:= bEnable_evac_mic,
	in_RefVAGF		:= VAGF, 
	in_RefVAGG		:= VAGG);
	

///////////////////////
// Pressure Ramp Test
///////////////////////
SIM_P1(	in_nType			:= E_CRYO_SENSOR_TYPE_PRESS.PKR_250, 
		in_lrBitsPerVolt	:= 3276.8, 
		in_lrPress			:= 777.0, 
		in_nPeriod			:= 10000);

// Start ramping from 100 to 0.0001 over 20 sec.
IF bStartRamp	THEN
	bStartRamp	:= FALSE;
	SIM_P1.M_SetValue(100.0);
	SIM_P1.M_RampTo(0.0001,20000);
END_IF
	
// Actuator test
actuator();
	
//
// FB_CRYO_ACTUATOR_CMD test.
//
// Allow only OPEN command for Valve2
cmdValve2.M_SetPermissions(in_bPermitOn := TRUE, in_bPermitOff := FALSE);
// Handling of Valve2 command with active interlock.
cmdValve2(in_bEnable := bEnable_Valve2, in_bInterlock := TRUE);	

Valve1(in_bEnable := bEnable_Valve1);		// Take system command as it is.
Valve2(in_bEnable := cmdValve2.out_bEnable);// Allow user to override system command.

//
// FB_CRYO_CMD_OVERRIDE Test
//
cmdOverrideTest(in_bEnable:=bEnable_OverrideTest);


//////////////////////////////
// Testing FB_CRYO_LN2_PRECOOL
//////////////////////////////
ln2_ctrl(
	in_bEnable		:= bEnable_ln2_ctrl, 
	in_lrTempK		:= SIM_ln2.lrTempK, 
	in_bTempValid	:= TRUE);

SIM_ln2(ln2Ref := ln2_ctrl);


/////////////////////////////////////////////
// Testing IO-Link FB_CRYO_SBG232 Flowmeter
/////////////////////////////////////////////
sbg232();

sbg232_sim(in_sName:='SBG232 SIM');
SIM_sbg232();

END_PROGRAM

// VISUs/GUIs/GUI_ATH2303M_EVAC_LAB
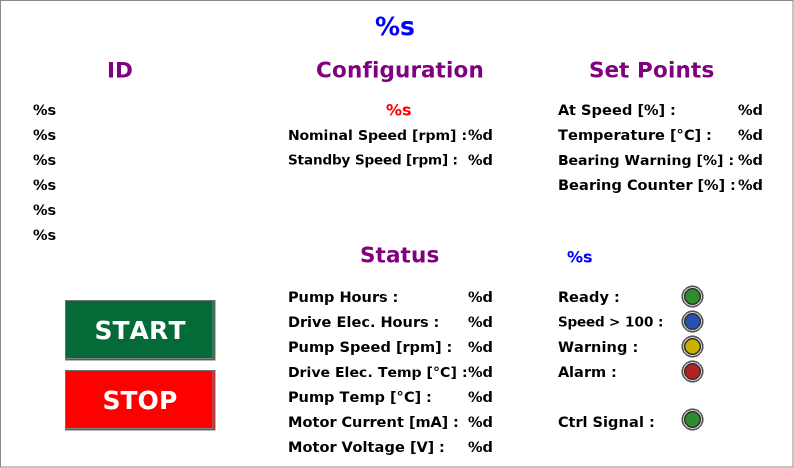
VISUALIZATION GUI_ATH2303M_EVAC_LAB  // 794x468
    Frame (0,0 794x468)
        shows GUI_TEMPLATE_ATH2303M(m_Instance := MAIN.evac_lab.tp, m_bEnable := MAIN.evac_lab.ctrl.bEnable_TP)
END_VISUALIZATION

// VISUs/GUIs/GUI_CMD_OVERRIDE
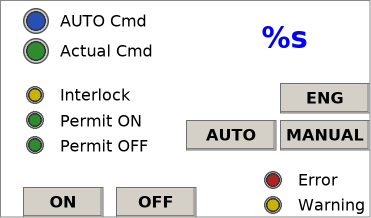
VISUALIZATION GUI_CMD_OVERRIDE  // 371x218
    Frame (0,0 371x218)
        shows GUI_TEMPLATE_CMD_OVERRIDE(m_Cmd := MAIN.cmdOverrideTest)
END_VISUALIZATION

// VISUs/GUIs/GUI_CPA
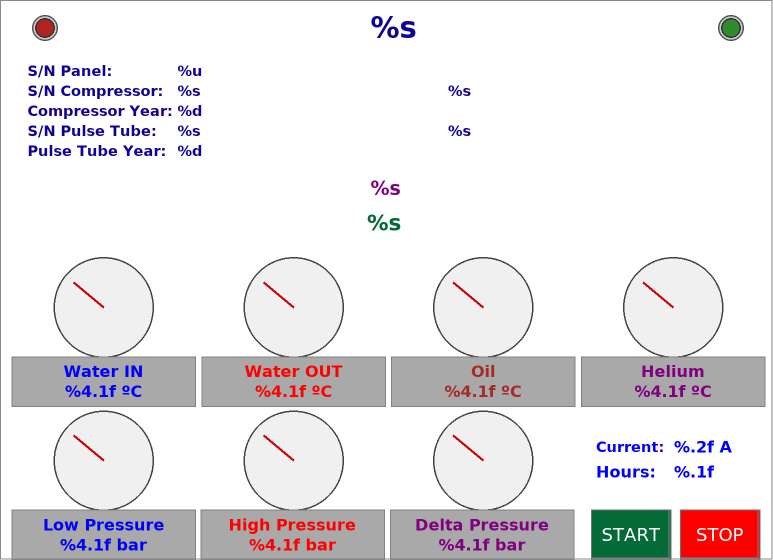
VISUALIZATION GUI_CPA  // 773x560
    Frame (0,0 773x560)
        shows GUI_TEMPLATE_CRYO_CPA(m_Instance := MAIN.Cryo_Ctrl.cpa)
END_VISUALIZATION

// VISUs/GUIs/GUI_CRYO
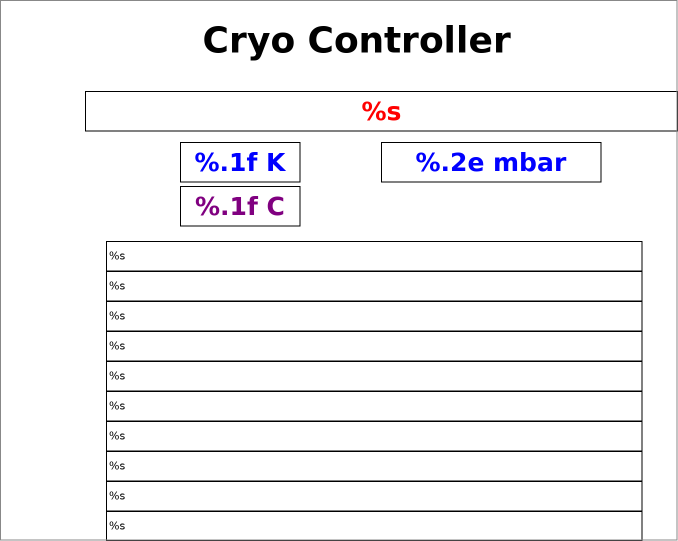
VISUALIZATION GUI_CRYO  // 678x541
    Rectangle (180,142 120x40), "%.1f K", text variable: MAIN.Cryo_Ctrl.Temp_ColdBench.stat.lrTempK
    Rectangle (180,186 120x40), "%.1f C", text variable: MAIN.Cryo_Ctrl.Temp_ColdBench.stat.lrTempC
    Rectangle (381,142 220x40), "%.2e mbar", text variable: MAIN.Cryo_Ctrl.Pressure_Cryo.stat.lrPressure
    Label (182,15 350x50), "Cryo Controller"
    Rectangle (85,91 593x40), "%s", text variable: MAIN.Cryo_Ctrl.stat.sState
    Rectangle (106,241 536x30), "%s", text variable: MAIN.Cryo_Ctrl.syslog.s9
    Rectangle (106,271 536x30), "%s", text variable: MAIN.Cryo_Ctrl.syslog.s8
    Rectangle (106,301 536x30), "%s", text variable: MAIN.Cryo_Ctrl.syslog.s7
    Rectangle (106,331 536x30), "%s", text variable: MAIN.Cryo_Ctrl.syslog.s6
    Rectangle (106,361 536x30), "%s", text variable: MAIN.Cryo_Ctrl.syslog.s5
    Rectangle (106,391 536x30), "%s", text variable: MAIN.Cryo_Ctrl.syslog.s4
    Rectangle (106,421 536x30), "%s", text variable: MAIN.Cryo_Ctrl.syslog.s3
    Rectangle (106,451 536x30), "%s", text variable: MAIN.Cryo_Ctrl.syslog.s2
    Rectangle (106,481 536x30), "%s", text variable: MAIN.Cryo_Ctrl.syslog.s1
    Rectangle (106,511 536x30), "%s", text variable: MAIN.Cryo_Ctrl.syslog.s0
END_VISUALIZATION

// VISUs/GUIs/GUI_CRYOTELGT
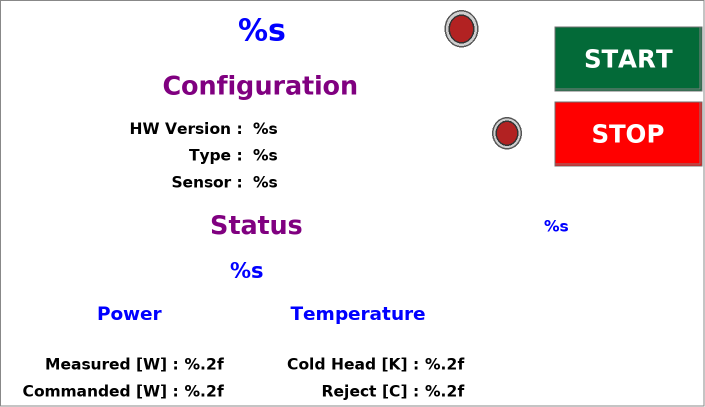
VISUALIZATION GUI_CRYOTELGT  // 705x407
    Frame (0,0 705x407)
        shows GUI_TEMPLATE_CRYOTELGT(m_Instance := MAIN.cooler, m_bEnable := MAIN.bEnable_cooler)
END_VISUALIZATION

// VISUs/GUIs/GUI_ECODRY_V01_EVAC_LAB
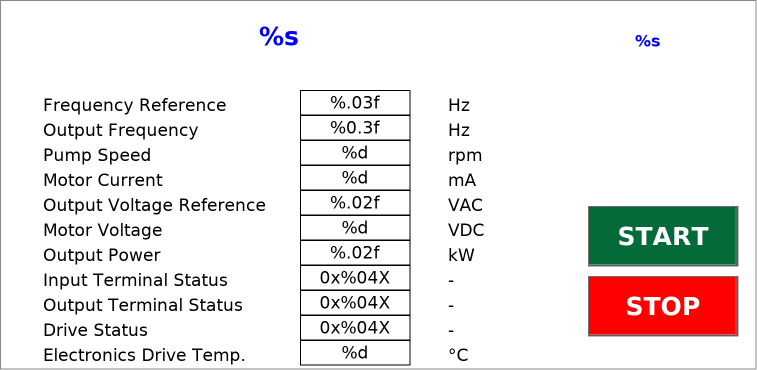
VISUALIZATION GUI_ECODRY_V01_EVAC_LAB  // 757x370
    Frame (0,0 757x370)
        shows GUI_TEMPLATE_ECODRY_V01(m_Instance := MAIN.evac_lab.rp, m_bEnable := MAIN.evac_lab.ctrl.bEnable_RP)
END_VISUALIZATION

// VISUs/GUIs/GUI_EVAC_LAB
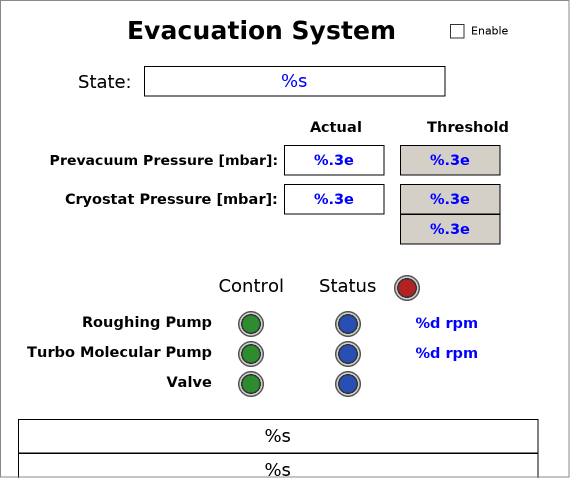
VISUALIZATION GUI_EVAC_LAB  // 570x478
    Frame (0,0 570x478)
        shows GUI_TEMPLATE_CRYO_EVAC_BASE(m_Instance := MAIN.evac_lab, m_bEnable := MAIN.bEnable_evac_lab)
END_VISUALIZATION

// VISUs/GUIs/GUI_EVAC_MICADO
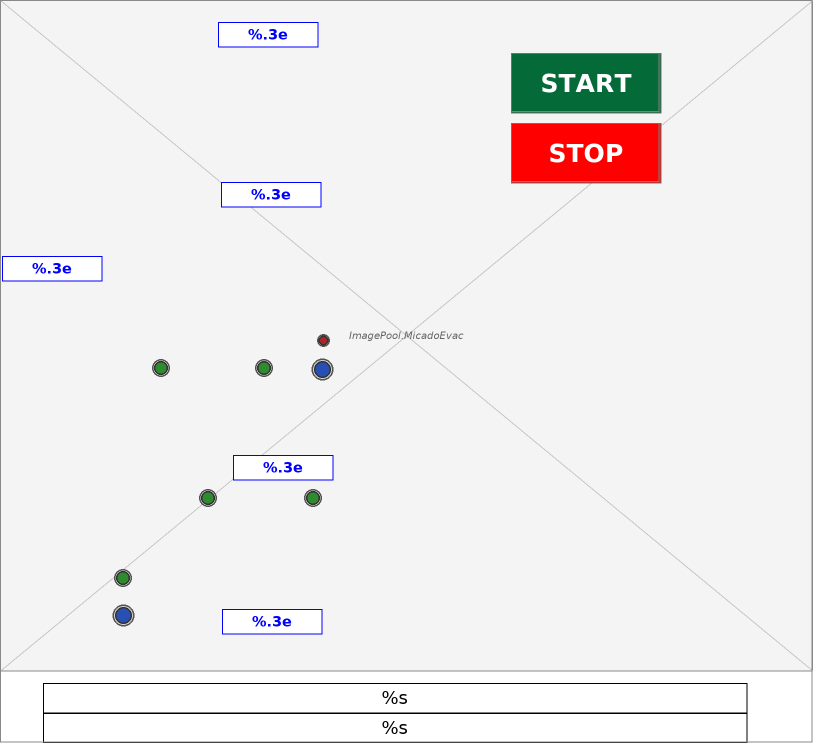
VISUALIZATION GUI_EVAC_MICADO  // 813x743
    Image (0,0 813x671), image: ImagePool.MicadoEvac
    Rectangle (222,609 100x25), "%.3e", text variable: MAIN.evac_micado.VAG1.stat.lrPressure
    Rectangle (233,455 100x25), "%.3e", text variable: MAIN.evac_micado.VAG2.stat.lrPressure
    Rectangle (2,256 100x25), "%.3e", text variable: MAIN.evac_micado.VAG3.stat.lrPressure
    Rectangle (218,22 100x25), "%.3e", text variable: MAIN.evac_micado.VAGF.stat.lrPressure
    Rectangle (221,182 100x25), "%.3e", text variable: MAIN.evac_micado.VAGG.stat.lrPressure
    Lamp1 (111,603 25x25), variable: MAIN.evac_micado.rp.stat.bReady, style: Lamp-Lamp1-Blue
    Lamp1 (310,357 25x25), tooltip "If ON, TMP pump is at its nominal speed, i.e. Ready.", variable: MAIN.evac_micado.tp.stat.bReady, style: Lamp-Lamp1-Blue
    Lamp1 (198,488 20x20), variable: MAIN.evac_micado.PVV1.stat.bActON, style: Lamp-Lamp1-Green
    Lamp1 (303,488 20x20), variable: MAIN.evac_micado.PVV2.stat.bActON, style: Lamp-Lamp1-Green
    Lamp1 (151,358 20x20), variable: MAIN.evac_micado.PVV3.stat.bActON, style: Lamp-Lamp1-Green
    Lamp1 (254,358 20x20), variable: MAIN.evac_micado.PVV4.stat.bActON, style: Lamp-Lamp1-Green
    Lamp1 (113,568 20x20), variable: MAIN.evac_micado.GBV.stat.bActON, style: Lamp-Lamp1-Green
    Rectangle (43,683 704x30), "%s", text variable: MAIN.evac_micado.stat.sErrorText
    Rectangle (43,713 704x30), "%s", text variable: MAIN.evac_micado.stat.sStatus
    Button (511,53 150x60), "START"
        OnMouseClick: execute { MAIN.bEnable_evac_mic := TRUE; }
    Button (511,123 150x60), "STOP"
        OnMouseClick: execute { MAIN.bEnable_evac_mic := FALSE; }
    Lamp1 (316,333 15x15), tooltip "If ON, TMP pump is still spinning.", variable: MAIN.evac_micado.tp.stat.bSpeed100, style: Lamp-Lamp1-Red
END_VISUALIZATION

// VISUs/GUIs/GUI_EVAC_PDS
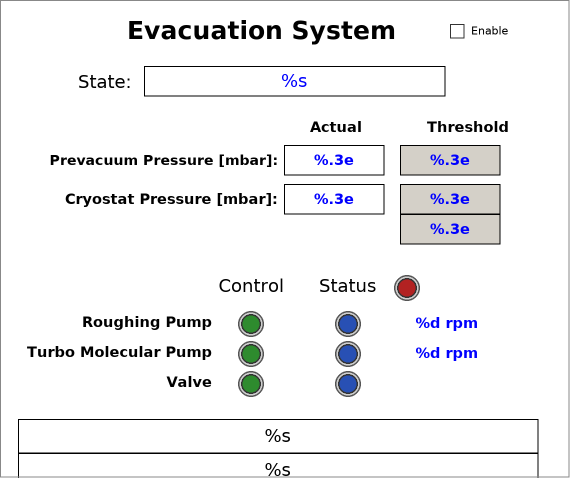
VISUALIZATION GUI_EVAC_PDS  // 570x478
    Frame (0,0 570x478)
        shows GUI_TEMPLATE_CRYO_EVAC_BASE(m_Instance := MAIN.evac_pds, m_bEnable := MAIN.bEnable_evac_pds)
END_VISUALIZATION

// VISUs/GUIs/GUI_HIPACE_30_EVAC_PDS
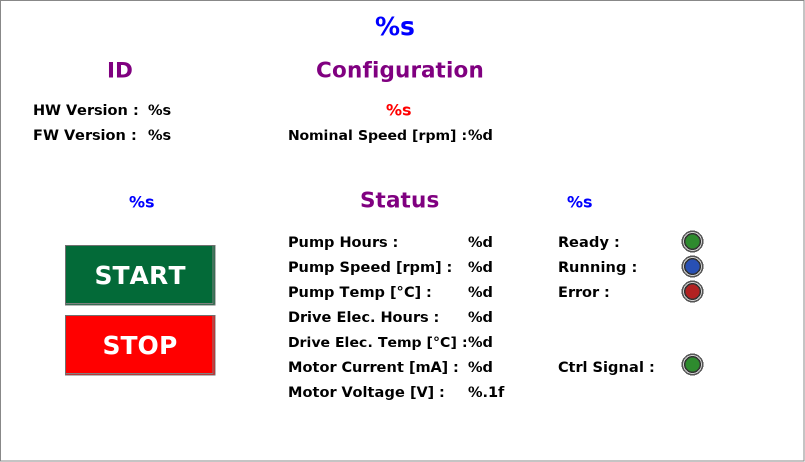
VISUALIZATION GUI_HIPACE_30_EVAC_PDS  // 805x462
    Frame (0,0 805x462)
        shows GUI_TEMPLATE_HIPACE_30(m_Instance := MAIN.evac_pds.tp, m_bEnable := MAIN.evac_pds.ctrl.bEnable_TP)
END_VISUALIZATION

// VISUs/GUIs/GUI_IRATEC
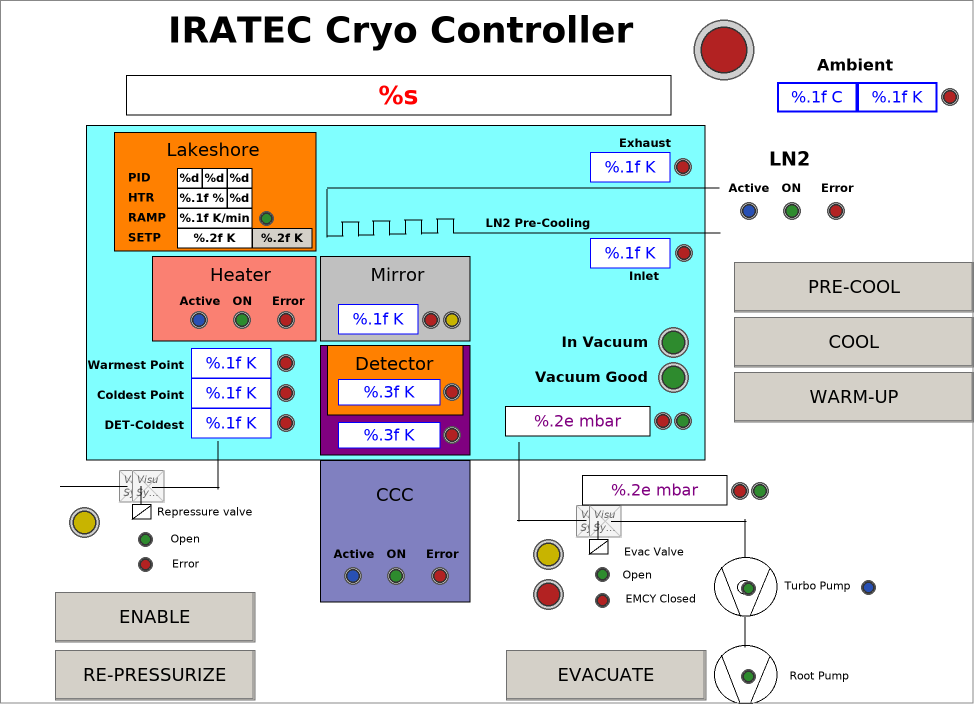
VISUALIZATION GUI_IRATEC  // 974x704
    RoundedRectangle (86,125 619x335)
    Group (327,188 393x50)
        Line (392,0) (0,0)
        Line (0,49) (0,1)
        Line (16,48) (0,48)
        Line (15,34) (15,48)
        Line (32,34) (14,34)
        Line (31,34) (31,48)
        Line (47,47) (31,47)
        Line (46,33) (46,47)
        Line (63,33) (45,33)
        Line (62,33) (62,47)
        Line (79,46) (63,46)
        Line (78,32) (78,46)
        Line (95,32) (77,32)
        Line (94,32) (94,46)
        Line (111,45) (95,45)
        Line (110,31) (110,45)
        Line (127,31) (109,31)
        Line (126,31) (126,45)
        Line (393,45) (126,45)
        Label (136,20 150x30), "LN2 Pre-Cooling"
    Group (714,557 63x59)
        Ellipse (0,0 63x59)
        Ellipse (23,23 15x14)
        Line (7,10) (26,59)
        Line (36,59) (56,11)
    Group (714,645 63x59)
        Ellipse (0,0 63x59)
        Line (7,10) (26,59)
        Line (36,59) (56,11)
    Line (745,647) (745,617)
    Image (576,505 32x32), image: VisuSymbols.Symbols.TriangleRight
    Group (589,505 32x49)
        Image (0,0 32x32), image: VisuSymbols.Symbols.TriangleLeft
        Rectangle (0,34 19x15)
        Line (0,49) (19,35)
        Line (9,34) (9,16)
    Line (745,557) (745,519)
    Line (611,521) (746,521)
    Line (517,520) (586,520)
    Line (519,521) (519,442)
    Rectangle (582,475 145x30), "%.2e mbar", text variable: MAIN.Cryo_Ctrl.Pressure_Evac.stat.lrPressure
    Rectangle (505,406 145x30), "%.2e mbar", text variable: MAIN.Cryo_Ctrl.Pressure_Cryo.stat.lrPressure
    Lamp1 (737,668 23x17), variable: MAIN.Cryo_Ctrl.EvacSys.stat.bRootPumpON, style: Lamp-Lamp1-Green
    Lamp1 (591,566 23x17), variable: MAIN.Cryo_Ctrl.EvacSys.stat.bValveOpen, style: Lamp-Lamp1-Green
    Image (119,470 32x32), image: VisuSymbols.Symbols.TriangleRight
    Group (132,470 32x49)
        Image (0,0 32x32), image: VisuSymbols.Symbols.TriangleLeft
        Rectangle (0,34 19x15)
        Line (0,49) (19,35)
        Line (9,34) (9,16)
    Lamp1 (134,531 23x17), variable: MAIN.Cryo_Ctrl.RepressValve.stat.bActON, style: Lamp-Lamp1-Green
    Line (218,489) (218,441)
    Line (152,487) (219,487)
    Line (60,486) (127,486)
    Label (130,497 150x30), "Repressure valve"
    Label (610,560 55x30), "Open"
    Lamp1 (656,360 35x35), variable: MAIN.Cryo_Ctrl.stat.bGoodVacuum, style: Lamp-Lamp1-Green
    Label (536,362 115x30), "Vacuum Good"
    Label (536,327 115x30), "In Vacuum"
    Lamp1 (656,325 35x35), variable: MAIN.Cryo_Ctrl.stat.bInVacuum, style: Lamp-Lamp1-Green
    Lamp1 (591,592 23x17), variable: MAIN.Cryo_Ctrl.EvacSys.stat.bEmergency, style: Lamp-Lamp1-Red
    Label (609,537 90x30), "Evac Valve"
    Label (614,584 94x30), "EMCY Closed"
    Lamp1 (737,580 23x17), variable: MAIN.Cryo_Ctrl.EvacSys.stat.bTurboPumpON, style: Lamp-Lamp1-Green
    Label (779,661 81x30), "Root Pump"
    Label (777,571 81x30), "Turbo Pump"
    Lamp1 (857,579 23x17), tooltip "Turbo Pump Ready", variable: MAIN.Cryo_Ctrl.EvacSys.stat.bTurboPump10min, style: Lamp-Lamp1-Blue
    Button (506,650 200x50), "EVACUATE", input disabled if: MAIN.Cryo_Ctrl.ctrl.bEnable_RepressSys=TRUE OR MAIN.Cryo_Ctrl.RepressValve.stat.bActON=TRUE
        toggle MAIN.Cryo_Ctrl.ctrl.bEnable_Evac
    Lamp1 (134,556 23x17), variable: MAIN.Cryo_Ctrl.RepressValve.stat.bError, style: Lamp-Lamp1-Red
    Label (158,524 55x30), "Open"
    Label (158,549 55x30), "Error"
    Button (55,592 200x50), "ENABLE", input disabled if: MAIN.Cryo_Ctrl.ctrl.bSafe_Repress=0
        toggle MAIN.Cryo_Ctrl.ctrl.bEnable_RepressSys
    Lamp1 (689,15 70x70), variable: MAIN.Cryo_Ctrl.stat.bError, invisible if: MAIN.Cryo_Ctrl.stat.bError = 0, style: Lamp-Lamp1-Red
    Rectangle (590,238 80x30), "%.1f K", text variable: MAIN.Cryo_Ctrl.Temp_LN2_Inlet.stat.lrTempK
    Rectangle (590,152 80x30), "%.1f K", text variable: MAIN.Cryo_Ctrl.Temp_LN2_Exhaust.stat.lrTempK
    Lamp1 (531,537 35x35), tooltip "If ON, system is enabled", variable: MAIN.Cryo_Ctrl.EvacSys.stat.bEnabled, style: Lamp-Lamp1-Yellow
    Lamp1 (67,505 35x35), tooltip "If ON, system is enabled", variable: MAIN.Cryo_Ctrl.ctrl.bEnable_RepressSys, style: Lamp-Lamp1-Yellow
    Group (716,144 150x77)
        Label (0,29 150x30), "Active ON Error"
        Lamp1 (23,57 20x20), variable: MAIN.Cryo_Ctrl.LN2.stat.bActive, style: Lamp-Lamp1-Blue
        Lamp1 (66,57 20x20), variable: MAIN.Cryo_Ctrl.LN2.stat.bActON, style: Lamp-Lamp1-Green
        Lamp1 (110,57 20x20), variable: MAIN.Cryo_Ctrl.LN2.stat.bError, style: Lamp-Lamp1-Red
        Label (36,0 75x30), "LN2"
    Lamp1 (531,577 35x35), tooltip "If ON, Evacuation System is in ERROR state.", variable: MAIN.Cryo_Ctrl.EvacSys.stat.bError, style: Lamp-Lamp1-Red
    Lamp1 (730,481 20x20), tooltip "Warning if reading is not valid", variable: NOT MAIN.Cryo_Ctrl.EvacSys.in_Pressure_Evac.bValid, style: Lamp-Lamp1-Red
    Group (320,460 151x142)
        Rectangle (0,0 150x142), "CCC"
        Lamp1 (23,106 20x20), tooltip "CCC Control is Enabled/Active", variable: MAIN.Cryo_Ctrl.CCC.stat.bActive, style: Lamp-Lamp1-Blue
        Lamp1 (66,106 20x20), tooltip "CCC is ON", variable: MAIN.Cryo_Ctrl.CCC.stat.bActON, style: Lamp-Lamp1-Green
        Lamp1 (110,106 20x20), variable: MAIN.Cryo_Ctrl.CCC.stat.bError, style: Lamp-Lamp1-Red
        Label (1,79 150x30), "Active ON Error"
    Label (602,128 86x30), "Exhaust"
    Label (601,261 86x30), "Inlet"
    Lamp1 (673,157 20x20), tooltip "Warning if reading is not valid", variable: NOT MAIN.Cryo_Ctrl.Temp_LN2_Exhaust.stat.bValid, style: Lamp-Lamp1-Red
    Lamp1 (674,243 20x20), tooltip "Warning if reading is not valid", variable: NOT MAIN.Cryo_Ctrl.Temp_LN2_Inlet.stat.bValid, style: Lamp-Lamp1-Red
    Lamp1 (653,411 20x20), tooltip "Warning if reading is not valid", variable: NOT MAIN.Cryo_Ctrl.Pressure_Cryo.stat.bValid, style: Lamp-Lamp1-Red
    Button (55,650 200x50), "RE-PRESSURIZE", input disabled if: MAIN.Cryo_Ctrl.ctrl.bEnable_RepressSys=0
        toggle MAIN.Cryo_Ctrl.ctrl.bEnable_RepressCtrl
    Button (734,262 240x50), "PRE-COOL", input disabled if: MAIN.Cryo_Ctrl.ctrl.bSafe_Precool = 0
        toggle MAIN.Cryo_Ctrl.ctrl.bEnable_Precool
    Button (734,317 240x50), "COOL", input disabled if: MAIN.Cryo_Ctrl.ctrl.bSafe_Cooling=0
        toggle MAIN.Cryo_Ctrl.ctrl.bEnable_Cool
    Button (734,372 240x50), "WARM-UP", input disabled if: MAIN.Cryo_Ctrl.ctrl.bSafe_Warmup=0
        toggle MAIN.Cryo_Ctrl.ctrl.bEnable_Warmup
    Label (152,5 498x50), "IRATEC Cryo Controller"
    Rectangle (126,75 545x40), "%s", text variable: MAIN.Cryo_Ctrl.stat.sState
    Group (152,256 165x85)
        Rectangle (0,0 164x85)
        Label (15,30 150x30), "Active ON Error"
        Lamp1 (37,54 20x20), tooltip "Heater Control is Enabled/Active", variable: MAIN.Cryo_Ctrl.Heater.stat.bActive, style: Lamp-Lamp1-Blue
        Lamp1 (80,54 20x20), tooltip "Heater is ON", variable: MAIN.Cryo_Ctrl.Heater.stat.bActON, style: Lamp-Lamp1-Green
        Lamp1 (124,54 20x20), variable: MAIN.Cryo_Ctrl.Heater.stat.bError, style: Lamp-Lamp1-Red
        Label (47,4 83x30), "Heater"
    Lamp1 (750,481 20x20), tooltip "Flag if reading is in sensor range", variable: MAIN.Cryo_Ctrl.EvacSys.in_Pressure_Evac.bInRange, style: Lamp-Lamp1-Green
    Lamp1 (673,411 20x20), tooltip "Flag if reading is in sensor range", variable: MAIN.Cryo_Ctrl.EvacSys.in_Pressure_Cryo.bInRange, style: Lamp-Lamp1-Green
    Label (92,380 95x30), "Coldest Point"
    Rectangle (191,378 80x30), "%.1f K", tooltip "Coldest point in the Cryostat", text variable: MAIN.Cryo_Ctrl.stat.lrLowestTempK
    Lamp1 (276,383 20x20), tooltip "Warning if reading is not valid", variable: NOT MAIN.Cryo_Ctrl.stat.bLowestTempValid, style: Lamp-Lamp1-Red
    Rectangle (191,408 80x30), "%.1f K", tooltip "Temperature difference between DET and the coldest point in the Cryostat", text variable: MAIN.Cryo_Ctrl.stat.lrDiffTempK
    Label (92,410 95x30), "DET-Coldest"
    Lamp1 (276,413 20x20), tooltip "Warning if reading is not valid", variable: NOT MAIN.Cryo_Ctrl.stat.bDiffTempValid, style: Lamp-Lamp1-Red
    Label (92,350 95x30), "Warmest Point"
    Rectangle (191,348 80x30), "%.1f K", tooltip "Warmest point in the Cryostat", text variable: MAIN.Cryo_Ctrl.stat.lrHighestTempK
    Lamp1 (276,353 20x20), tooltip "Warning if reading is not valid", variable: NOT MAIN.Cryo_Ctrl.stat.bHighestTempValid, style: Lamp-Lamp1-Red
    Rectangle (114,132 202x119)
    Label (160,135 106x30), "Lakeshore"
    Label (125,170 40x15), "PID"
    Label (125,190 40x15), "HTR"
    Label (125,210 40x15), "RAMP"
    Label (125,230 40x15), "SETP"
    Rectangle (177,168 25x20), "%d", text variable: MAIN.Cryo_Ctrl.Lakeshore.stat.nPID_P
    Rectangle (202,168 25x20), "%d", text variable: MAIN.Cryo_Ctrl.Lakeshore.stat.nPID_I
    Rectangle (227,168 25x20), "%d", text variable: MAIN.Cryo_Ctrl.Lakeshore.stat.nPID_D
    Rectangle (177,188 50x20), "%.1f %", tooltip "Heater Output [%]", text variable: MAIN.Cryo_Ctrl.Lakeshore.stat.lrHTR
    Rectangle (177,208 75x20), "%.1f K/min", tooltip "Heater Ramp Rate", text variable: MAIN.Cryo_Ctrl.Lakeshore.stat.lrRAMP_Rate
    Lamp1 (255,210 23x17), tooltip "Flag if Heater RAMP is On", variable: MAIN.Cryo_Ctrl.Lakeshore.stat.bRAMP_On, style: Lamp-Lamp1-Green
    Rectangle (177,228 75x20), "%.2f K", tooltip "SetPoint", text variable: MAIN.Cryo_Ctrl.Lakeshore.stat.lrSETP
    Rectangle (227,188 25x20), "%d", tooltip "Heater Range", text variable: MAIN.Cryo_Ctrl.Lakeshore.stat.nRANGE
    Group (320,256 150x85)
        Rectangle (0,0 150x85)
        Label (29,4 97x30), "Mirror"
        Rectangle (18,48 80x30), "%.1f K", text variable: MAIN.Cryo_Ctrl.Temp_Mirror.stat.lrTempK
        Lamp1 (101,54 20x20), tooltip "Warning if reading is not valid", variable: NOT MAIN.Cryo_Ctrl.Temp_Mirror.stat.bValid, style: Lamp-Lamp1-Red
        Lamp1 (122,54 20x20), tooltip "Warning if reading is underrange. PT100 cannot read below 73.15K (-200C).", variable: NOT MAIN.Cryo_Ctrl.Temp_Mirror.stat.bInRange, style: Lamp-Lamp1-Yellow
    Group (320,345 150x110)
        Rectangle (0,0 150x110)
        Rectangle (18,77 102x26), "%.3f K", tooltip "Heat Shield Temperature", text variable: MAIN.Cryo_Ctrl.Temp_HeatShield.stat.lrTempK
        Lamp1 (122,80 20x20), tooltip "Warning if reading is not valid", variable: NOT MAIN.Cryo_Ctrl.Temp_HeatShield.stat.bValid, style: Lamp-Lamp1-Red
    Group (327,345 136x70)
        Rectangle (0,0 136x70)
        Rectangle (11,34 102x26), "%.3f K", text variable: MAIN.Cryo_Ctrl.Temp_DET.stat.lrTempK
        Lamp1 (115,37 20x20), tooltip "Warning if reading is not valid", variable: NOT MAIN.Cryo_Ctrl.Temp_DET.stat.bValid, style: Lamp-Lamp1-Red
        Label (26,4 83x30), "Detector"
    Rectangle (252,228 60x20), "%.2f K", tooltip "Target SetPoint", text variable: MAIN.Cryo_Ctrl.Lakeshore.stat.lrSETP_Target
    Rectangle (857,82 80x30), "%.1f K", text variable: MAIN.Cryo_Ctrl.Temp_Ambient.stat.lrTempK
    Lamp1 (940,87 20x20), tooltip "Warning if reading is not valid", variable: NOT MAIN.Cryo_Ctrl.Temp_Ambient.stat.bValid, style: Lamp-Lamp1-Red
    Rectangle (777,82 80x30), "%.1f C", text variable: MAIN.Cryo_Ctrl.Temp_Ambient.stat.lrTempC
    Label (812,50 86x30), "Ambient"
END_VISUALIZATION

// VISUs/GUIs/GUI_MICADO_Valves
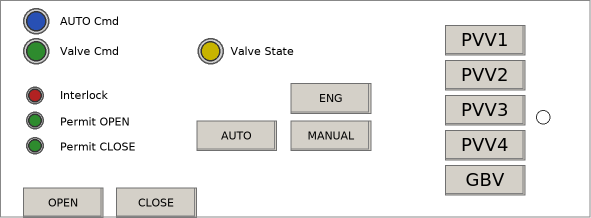
VISUALIZATION GUI_MICADO_Valves  // 591x218
    Frame (0,0 371x218)
        shows GUI_TEMPLATE_ACTUATOR_ENG(m_Cmd := MAIN.evac_micado.ptrVC[MAIN.evac_micado.guiValveIndex]^, m_Valve := MAIN.evac_micado.ptrV[MAIN.evac_micado.guiValveIndex]^)
    Button (445,25 80x30), "PVV1"
        OnMouseClick: execute { MAIN.evac_micado.guiValveIndex := 1; }
    Button (445,60 80x30), "PVV2"
        OnMouseClick: execute { MAIN.evac_micado.guiValveIndex := 2; }
    Button (445,95 80x30), "PVV3"
        OnMouseClick: execute { MAIN.evac_micado.guiValveIndex := 3; }
    Button (445,130 80x30), "PVV4"
        OnMouseClick: execute { MAIN.evac_micado.guiValveIndex := 4; }
    Button (445,165 80x30), "GBV"
        OnMouseClick: execute { MAIN.evac_micado.guiValveIndex := 5; }
    RadioButton (534,28 57x178), variable: MAIN.evac_micado.guiValveIndex-1
END_VISUALIZATION

// VISUs/GUIs/GUI_MVP030_EVAC_PDS
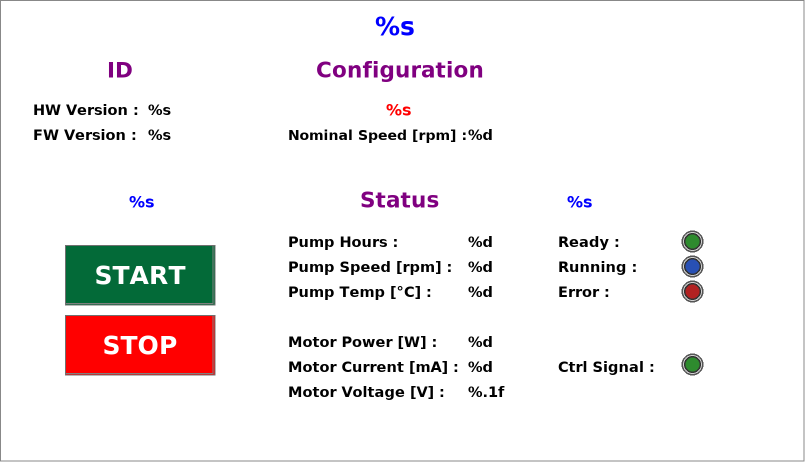
VISUALIZATION GUI_MVP030_EVAC_PDS  // 805x462
    Frame (0,0 805x462)
        shows GUI_TEMPLATE_MVP030(m_Instance := MAIN.evac_pds.rp, m_bEnable := MAIN.evac_pds.ctrl.bEnable_RP)
END_VISUALIZATION

// VISUs/GUIs/GUI_P2_OVERRIDE
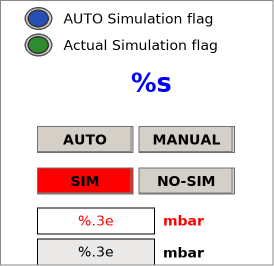
VISUALIZATION GUI_P2_OVERRIDE  // 274x266
    Frame (0,0 274x266)
        shows GUI_TEMPLATE_PRESS_OVERRIDE(m_Cmd := MAIN.pressOR_P1, m_Press := MAIN.P1)
END_VISUALIZATION

// VISUs/GUIs/GUI_Pressures
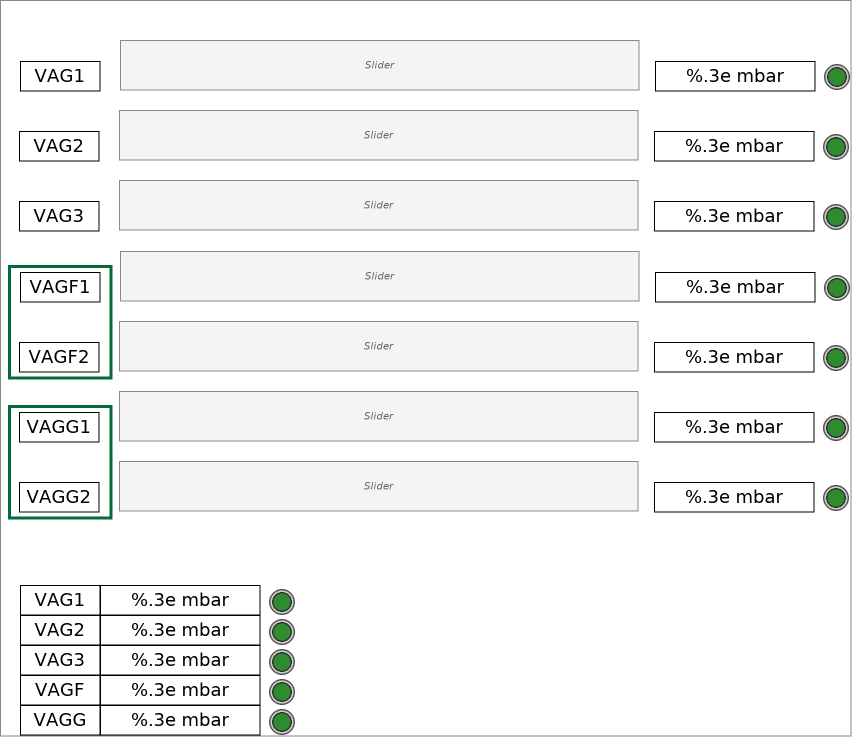
VISUALIZATION GUI_Pressures  // 852x737
    Slider (120,40 519x50), variable: MAIN.q_nVAG1, scale 0..35000
    Rectangle (20,61 80x30), "VAG1"
    Rectangle (655,61 160x30), "%.3e mbar", text variable: MAIN.evac_micado.VAG1.stat.lrPressure
    Lamp1 (822,62 30x30), variable: MAIN.evac_micado.VAG1.stat.bValid, style: Lamp-Lamp1-Green
    Slider (119,110 519x50), variable: MAIN.q_nVAG2, scale 0..35000
    Rectangle (19,131 80x30), "VAG2"
    Rectangle (654,131 160x30), "%.3e mbar", text variable: MAIN.evac_micado.VAG2.stat.lrPressure
    Lamp1 (821,132 30x30), variable: MAIN.evac_micado.VAG2.stat.bValid, style: Lamp-Lamp1-Green
    Slider (119,180 519x50), variable: MAIN.q_nVAG3, scale 0..35000
    Rectangle (19,201 80x30), "VAG3"
    Rectangle (654,201 160x30), "%.3e mbar", text variable: MAIN.evac_micado.VAG3.stat.lrPressure
    Lamp1 (821,202 30x30), variable: MAIN.evac_micado.VAG3.stat.bValid, style: Lamp-Lamp1-Green
    Slider (120,251 519x50), variable: MAIN.q_nVAGF1, scale 0..35000
    Rectangle (20,272 80x30), "VAGF1"
    Rectangle (655,272 160x30), "%.3e mbar", text variable: MAIN.sensor_VAGF1.stat.lrPressure
    Lamp1 (822,273 30x30), variable: MAIN.sensor_VAGF1.stat.bValid, style: Lamp-Lamp1-Green
    Slider (119,321 519x50), variable: MAIN.q_nVAGF2, scale 0..35000
    Rectangle (19,342 80x30), "VAGF2"
    Rectangle (654,342 160x30), "%.3e mbar", text variable: MAIN.sensor_VAGF2.stat.lrPressure
    Lamp1 (821,343 30x30), variable: MAIN.sensor_VAGF2.stat.bValid, style: Lamp-Lamp1-Green
    Slider (119,391 519x50), variable: MAIN.q_nVAGG1, scale 0..35000
    Rectangle (19,412 80x30), "VAGG1"
    Rectangle (654,412 160x30), "%.3e mbar", text variable: MAIN.sensor_VAGG1.stat.lrPressure
    Lamp1 (821,413 30x30), variable: MAIN.sensor_VAGG1.stat.bValid, style: Lamp-Lamp1-Green
    Slider (119,461 519x50), variable: MAIN.q_nVAGG2, scale 0..35000
    Rectangle (19,482 80x30), "VAGG2"
    Rectangle (654,482 160x30), "%.3e mbar", text variable: MAIN.sensor_VAGG2.stat.lrPressure
    Lamp1 (821,483 30x30), variable: MAIN.sensor_VAGG2.stat.bValid, style: Lamp-Lamp1-Green
    Rectangle (20,585 80x30), "VAG1"
    Rectangle (20,615 80x30), "VAG2"
    Rectangle (20,645 80x30), "VAG3"
    Rectangle (100,585 160x30), "%.3e mbar", text variable: MAIN.evac_micado.VAG1.stat.lrPressure
    Lamp1 (267,587 30x30), variable: MAIN.evac_micado.VAG1.stat.bValid, style: Lamp-Lamp1-Green
    Rectangle (100,615 160x30), "%.3e mbar", text variable: MAIN.evac_micado.VAG2.stat.lrPressure
    Lamp1 (267,617 30x30), variable: MAIN.evac_micado.VAG2.stat.bValid, style: Lamp-Lamp1-Green
    Rectangle (100,645 160x30), "%.3e mbar", text variable: MAIN.evac_micado.VAG3.stat.lrPressure
    Lamp1 (267,647 30x30), variable: MAIN.evac_micado.VAG3.stat.bValid, style: Lamp-Lamp1-Green
    Rectangle (20,675 80x30), "VAGF"
    Rectangle (100,675 160x30), "%.3e mbar", text variable: MAIN.evac_micado.VAGF.stat.lrPressure
    Lamp1 (267,677 30x30), variable: MAIN.evac_micado.VAGF.stat.bValid, style: Lamp-Lamp1-Green
    Rectangle (20,705 80x30), "VAGG"
    Rectangle (100,705 160x30), "%.3e mbar", text variable: MAIN.evac_micado.VAGG.stat.lrPressure
    Lamp1 (267,707 30x30), variable: MAIN.evac_micado.VAGG.stat.bValid, style: Lamp-Lamp1-Green
    Rectangle (8,265 104x114)
    Rectangle (8,405 104x114)
END_VISUALIZATION

// VISUs/GUIs/GUI_PVV1_CMD
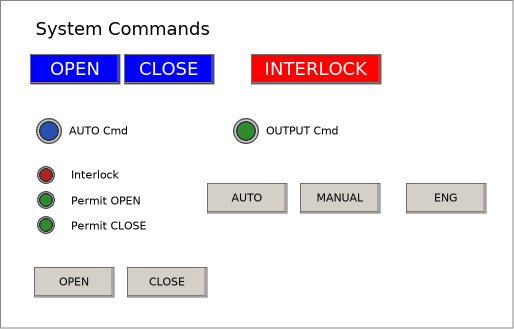
VISUALIZATION GUI_PVV1_CMD  // 514x329
    Frame (11,105 503x224)
        shows GUI_TEMPLATE_ACTUATOR_CMD(m_Instance := MAIN.cmdPVV1)
    Button (30,54 90x30), "OPEN", tooltip "Set External System command to OPEN"
        OnMouseClick: execute { MAIN.bCmdPVV1 := TRUE; }
    Button (124,54 90x30), "CLOSE", tooltip "Set External System command to CLOSE"
        OnMouseClick: execute { MAIN.bCmdPVV1 := FALSE; }
    Rectangle (33,14 180x30), "System Commands"
    Button (251,54 130x30), "INTERLOCK", tooltip "Toggle External System INTERLOCK"
        toggle MAIN.bIntlkPVV1
        OnMouseClick: execute { MAIN.bCmdPVV1 := TRUE; }
END_VISUALIZATION

// VISUs/GUIs/GUI_SBG232
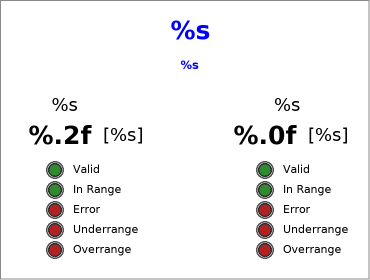
VISUALIZATION GUI_SBG232  // 370x280
    Frame (0,0 370x280)
        shows GUI_TEMPLATE_SBG232(m_Instance := MAIN.sbg232)
END_VISUALIZATION

// VISUs/GUIs/GUI_SBG232_SIM
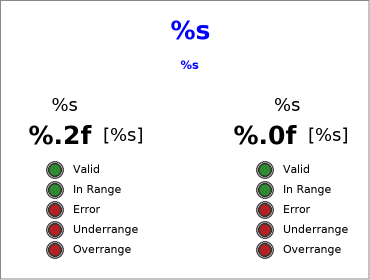
VISUALIZATION GUI_SBG232_SIM  // 370x280
    Frame (0,0 370x280)
        shows GUI_TEMPLATE_SBG232(m_Instance := MAIN.sbg232_sim)
END_VISUALIZATION

// VISUs/GUIs/GUI_T2_OVERRIDE
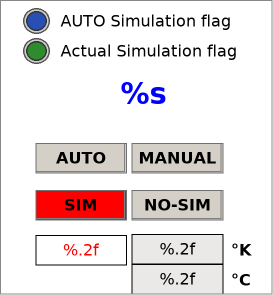
VISUALIZATION GUI_T2_OVERRIDE  // 273x295
    Frame (0,0 273x295)
        shows GUI_TEMPLATE_TEMP_OVERRIDE(m_Cmd := MAIN.tempOR_T2, m_Temp := MAIN.T2)
END_VISUALIZATION

// VISUs/Templates/GUI_TEMPLATE_ACTUATOR_CMD
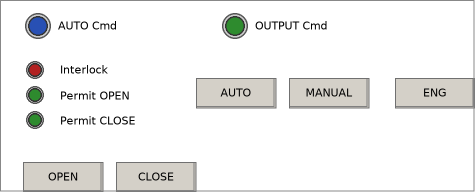
VISUALIZATION GUI_TEMPLATE_ACTUATOR_CMD  // 475x192
VAR_IN_OUT
	m_Instance:	FB_CRYO_ACTUATOR_CMD;
END_VAR
    Lamp1 (25,60 20x20), variable: m_Instance.in_bInterlock, style: Lamp-Lamp1-Red
    Lamp1 (25,85 20x20), variable: m_Instance.bPermitOn, style: Lamp-Lamp1-Green
    Lamp1 (25,110 20x20), variable: m_Instance.bPermitOff, style: Lamp-Lamp1-Green
    Rectangle (57,55 83x30), "Interlock"
    Rectangle (57,81 83x30), "Permit OPEN"
    Rectangle (57,106 83x30), "Permit CLOSE"
    Button (23,162 80x30), "OPEN", colour toggle: (m_Instance.bPermitOn AND NOT m_Instance.bAutoMode) OR m_Instance.bEngMode, input disabled if: m_Instance.bDisableBtnOn
        OnMouseClick: execute { m_Instance.bManualCmd := TRUE; m_Instance.bManualExecute := TRUE; }
    Lamp1 (220,11 30x30), variable: m_Instance.out_Enable, style: Lamp-Lamp1-Green
    Rectangle (252,11 83x30), "OUTPUT Cmd"
    Button (196,78 80x30), "AUTO", colour toggle: m_Instance.bAutoMode, input disabled if: m_Instance.bAutoMode OR m_Instance.bEngMode
        OnMouseClick: execute { m_Instance.bAutoMode := TRUE; }
    Button (289,78 80x30), "MANUAL", colour toggle: NOT m_Instance.bAutoMode, input disabled if: NOT m_Instance.bAutoMode AND NOT_IDLE m_Instance.bEngMode
        OnMouseClick: execute { m_Instance.bAutoMode := FALSE; }
    Button (116,162 80x30), "CLOSE", colour toggle: (m_Instance.bPermitOff AND NOT m_Instance.bAutoMode) OR m_Instance.bEngMode, input disabled if: m_Instance.bDisableBtnOff
        OnMouseClick: execute { m_Instance.bManualCmd := FALSE; m_Instance.bManualExecute := TRUE; }
    Button (395,78 80x30), "ENG", tooltip "Engineering / Commissioning Mode", colour toggle: m_Instance.bEngMode, input disabled if: m_Instance.bAutoMode
        toggle m_Instance.bEngMode
    Lamp1 (23,11 30x30), variable: m_Instance.in_bEnable, style: Lamp-Lamp1-Blue
    Rectangle (55,11 83x30), "AUTO Cmd"
END_VISUALIZATION

// VISUs/Templates/GUI_TEMPLATE_ACTUATOR_ENG
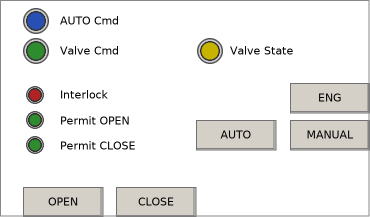
VISUALIZATION GUI_TEMPLATE_ACTUATOR_ENG  // 370x217
VAR_IN_OUT
	m_Cmd:		FB_CRYO_ACTUATOR_CMD;
	m_Valve:	FB_CRYO_VALVE_CTRL;
END_VAR
    Lamp1 (25,85 20x20), variable: m_Cmd.in_bInterlock, style: Lamp-Lamp1-Red
    Lamp1 (25,110 20x20), variable: m_Cmd.bPermitOn, style: Lamp-Lamp1-Green
    Lamp1 (25,135 20x20), variable: m_Cmd.bPermitOff, style: Lamp-Lamp1-Green
    Rectangle (57,80 83x30), "Interlock"
    Rectangle (57,106 83x30), "Permit OPEN"
    Rectangle (57,131 83x30), "Permit CLOSE"
    Button (23,187 80x30), "OPEN", colour toggle: (m_Cmd.bPermitOn AND NOT m_Cmd.bAutoMode) OR m_Cmd.bEngMode, input disabled if: m_Cmd.bDisableBtnOn
        OnMouseClick: execute { m_Cmd.bManualCmd := TRUE; m_Cmd.bManualExecute := TRUE; }
    Lamp1 (21,36 30x30), tooltip "Actual Valve command", variable: m_Cmd.out_bEnable, style: Lamp-Lamp1-Green
    Rectangle (57,36 83x30), "Valve Cmd"
    Button (196,120 80x30), "AUTO", colour toggle: m_Cmd.bAutoMode, input disabled if: m_Cmd.bAutoMode OR m_Cmd.bEngMode
        OnMouseClick: execute { m_Cmd.bAutoMode := TRUE; }
    Button (290,120 80x30), "MANUAL", colour toggle: NOT m_Cmd.bAutoMode, input disabled if: NOT m_Cmd.bAutoMode AND NOT m_Cmd.bEngMode
        OnMouseClick: execute { m_Cmd.bAutoMode := FALSE; }
    Button (116,187 80x30), "CLOSE", colour toggle: (m_Cmd.bPermitOff AND NOT m_Cmd.bAutoMode) OR m_Cmd.bEngMode, input disabled if: m_Cmd.bDisableBtnOff
        OnMouseClick: execute { m_Cmd.bManualCmd := FALSE; m_Cmd.bManualExecute := TRUE; }
    Button (290,83 80x30), "ENG", tooltip "Engineering / Commissioning Mode", colour toggle: m_Cmd.bEngMode, input disabled if: m_Cmd.bAutoMode
        toggle m_Cmd.bEngMode
    Lamp1 (21,6 30x30), tooltip "Command coming from the Control System", variable: m_Cmd.in_bEnable, style: Lamp-Lamp1-Blue
    Rectangle (57,6 83x30), "AUTO Cmd"
    Lamp1 (195,36 30x30), tooltip "Valve state: ON=OPEN, OFF=CLOSED", variable: m_Valve.stat.bActON, style: Lamp-Lamp1-Yellow
    Rectangle (227,36 83x30), "Valve State"
END_VISUALIZATION

// VISUs/Templates/GUI_TEMPLATE_ATH2303M
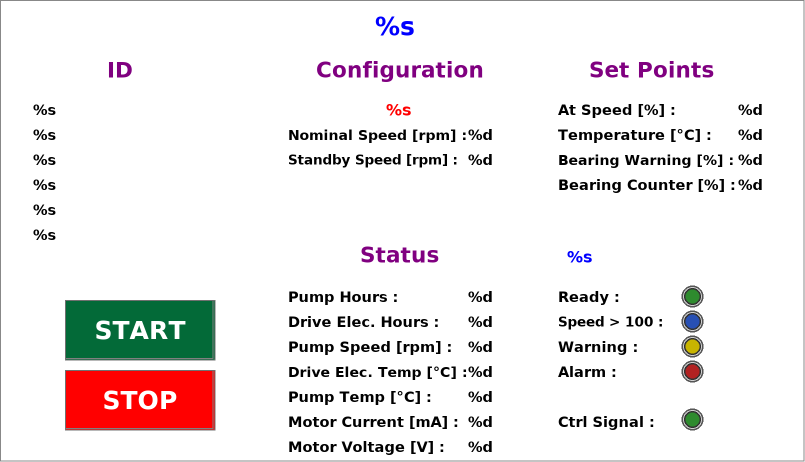
VISUALIZATION GUI_TEMPLATE_ATH2303M  // 805x462
VAR_IN_OUT
	m_Instance:	FB_CRYO_PUMP_ATH2303M;
	m_bEnable:	BOOL;	// Flag to start/stop the pump
END_VAR
    Rectangle (45,55 150x30), "ID"
    Rectangle (310,55 180x30), "Configuration"
    Rectangle (325,240 150x30), "Status"
    Lamp1 (680,284 25x25), tooltip "OK for Process, i.e. speed ≥ nominal speed", variable: m_Instance.stat.bReady, style: Lamp-Lamp1-Green
    Lamp1 (680,309 25x25), tooltip "pump speed > 100 rpm", variable: m_Instance.stat.bSpeed100, style: Lamp-Lamp1-Blue
    Lamp1 (680,334 25x25), tooltip "presence of a warning", variable: m_Instance.stat.bWarning, style: Lamp-Lamp1-Yellow
    Lamp1 (680,359 25x25), tooltip "presence of an alarm", variable: m_Instance.stat.bAlarm, style: Lamp-Lamp1-Red
    Rectangle (555,282 110x30), "Ready :"
    Rectangle (555,307 110x30), "Speed > 100 :"
    Rectangle (555,332 110x30), "Warning :"
    Rectangle (555,357 110x30), "Alarm :"
    Rectangle (30,145 240x30), "%s", text variable: m_Instance.stat.sVer1
    Rectangle (30,170 240x30), "%s", text variable: m_Instance.stat.sVer2
    Rectangle (30,195 240x30), "%s", text variable: m_Instance.stat.sVer3
    Rectangle (30,220 240x30), "%s", text variable: m_Instance.stat.sVer4
    Rectangle (285,120 180x30), "Nominal Speed [rpm] :"
    Rectangle (285,145 180x30), "Standby Speed [rpm] :"
    Rectangle (285,282 180x30), "Pump Hours :"
    Rectangle (285,307 180x30), "Drive Elec. Hours :"
    Rectangle (577,55 150x30), "Set Points"
    Rectangle (555,95 180x30), "At Speed [%] :"
    Rectangle (555,120 180x30), "Temperature [°C] :"
    Rectangle (555,145 180x30), "Bearing Warning [%] :"
    Rectangle (555,170 180x30), "Bearing Counter [%] :"
    Rectangle (735,95 70x30), "%d", text variable: m_Instance.stat.nSetPoint_AtSpeed
    Rectangle (735,120 70x30), "%d", text variable: m_Instance.stat.nSetPoint_Temp
    Rectangle (735,145 70x30), "%d", text variable: m_Instance.stat.nSetPoint_BearingWarn
    Rectangle (735,170 70x30), "%d", text variable: m_Instance.stat.nSetPoint_BearingCounter
    Rectangle (465,120 70x30), "%d", text variable: m_Instance.stat.nNominalSpeed
    Rectangle (465,145 70x30), "%d", text variable: m_Instance.stat.nStandbySpeed
    Rectangle (465,282 70x30), "%d", text variable: m_Instance.stat.nPumpHours
    Rectangle (465,307 70x30), "%d", text variable: m_Instance.stat.nElecHours
    Rectangle (285,332 180x30), "Pump Speed [rpm] :"
    Rectangle (465,332 70x30), "%d", text variable: m_Instance.stat.nPumpSpeed
    Rectangle (285,357 180x30), "Drive Elec. Temp [°C] :"
    Rectangle (465,357 70x30), "%d", text variable: m_Instance.stat.nElecTemp
    Rectangle (285,382 180x30), "Pump Temp [°C] :"
    Rectangle (465,382 70x30), "%d", text variable: m_Instance.stat.nPumpTemp
    Rectangle (285,407 180x30), "Motor Current [mA] :"
    Rectangle (465,407 70x30), "%d", text variable: m_Instance.stat.nMotorCurr
    Rectangle (285,432 180x30), "Motor Voltage [V] :"
    Rectangle (465,432 70x30), "%d", text variable: m_Instance.stat.nMotorVolt
    Rectangle (280,11 230x30), "%s", text variable: m_Instance.in_sName
    Rectangle (289,95 220x30), "%s", tooltip "Control Mode", text variable: m_Instance.stat.sCtrlMode
    Rectangle (30,95 240x30), "%s", text variable: m_Instance.stat.sIDN
    Rectangle (30,120 240x30), "%s", text variable: m_Instance.stat.sRDI
    Button (65,300 150x60), "START"
        OnMouseClick: execute { m_bEnable := TRUE; }
    Button (65,370 150x60), "STOP"
        OnMouseClick: execute { m_bEnable := FALSE; }
    Lamp1 (680,407 25x25), tooltip "If ON, control output signal is active.", variable: m_Instance.q_bStart, style: Lamp-Lamp1-Green
    Rectangle (555,407 110x30), "Ctrl Signal :"
    Rectangle (457,242 246x30), "%s", tooltip "Control Mode", text variable: m_Instance.stat.sPumpState
END_VISUALIZATION

// VISUs/Templates/GUI_TEMPLATE_CMD_OVERRIDE
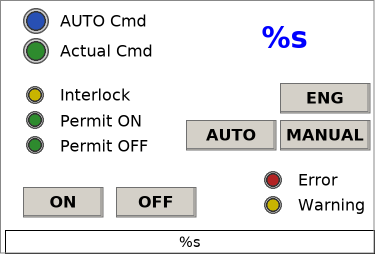
VISUALIZATION GUI_TEMPLATE_CMD_OVERRIDE  // 375x254
VAR_IN_OUT
	m_Cmd:		FB_CRYO_CMD_OVERRIDE;
END_VAR
    Lamp1 (25,85 20x20), variable: m_Cmd.out_bInterlock, style: Lamp-Lamp1-Yellow
    Lamp1 (25,110 20x20), variable: m_Cmd.bPermitOn, style: Lamp-Lamp1-Green
    Lamp1 (25,135 20x20), variable: m_Cmd.bPermitOff, style: Lamp-Lamp1-Green
    Rectangle (57,80 110x30), "Interlock"
    Rectangle (57,106 110x30), "Permit ON"
    Rectangle (57,131 110x30), "Permit OFF"
    Button (23,187 80x30), "ON", colour toggle: (m_Cmd.bPermitOn AND NOT m_Cmd.bAutoMode) OR m_Cmd.bEngMode, input disabled if: m_Cmd.bDisableBtnOn
        OnMouseClick: execute { m_Cmd.bManualCmd := TRUE; }
    Lamp1 (21,36 30x30), tooltip "Actual command going out", variable: m_Cmd.out_bEnable, style: Lamp-Lamp1-Green
    Rectangle (57,36 110x30), "Actual Cmd"
    Button (186,120 90x30), "AUTO", tooltip "Switch to AUTO Mode", colour toggle: m_Cmd.bAutoMode, input disabled if: m_Cmd.bAutoMode OR m_Cmd.bEngMode
        OnMouseClick: execute { m_Cmd.bAutoMode := TRUE; }
    Button (280,120 90x30), "MANUAL", tooltip "Switch to MANUAL Mode", colour toggle: NOT m_Cmd.bAutoMode, input disabled if: NOT m_Cmd.bAutoMode AND NOT m_Cmd.bEngMode
        OnMouseClick: execute { m_Cmd.bAutoMode := FALSE; }
    Button (116,187 80x30), "OFF", colour toggle: (m_Cmd.bPermitOff AND NOT m_Cmd.bAutoMode) OR m_Cmd.bEngMode, input disabled if: m_Cmd.bDisableBtnOff
        OnMouseClick: execute { m_Cmd.bManualCmd := FALSE; }
    Button (280,83 90x30), "ENG", tooltip "Toggle Engineering Mode", colour toggle: m_Cmd.bEngMode, input disabled if: m_Cmd.bAutoMode
        toggle m_Cmd.bEngMode
    Lamp1 (21,6 30x30), tooltip "Command coming from the Control System", variable: m_Cmd.in_bEnable, style: Lamp-Lamp1-Blue
    Rectangle (57,6 110x30), "AUTO Cmd"
    Rectangle (5,230 370x24), "%s", text variable: m_Cmd.out_sStatus
    Lamp1 (263,170 20x20), tooltip "If ON, there is an error in the SW implementation of permission handling.", variable: m_Cmd.out_bError, style: Lamp-Lamp1-Red
    Rectangle (295,165 75x30), "Error"
    Lamp1 (263,195 20x20), tooltip "If ON, ENG command is not safe!", variable: m_Cmd.out_bWarning, style: Lamp-Lamp1-Yellow
    Rectangle (295,190 75x30), "Warning"
    Rectangle (210,17 150x41), "%s", text variable: m_Cmd.out_sMode
END_VISUALIZATION

// VISUs/Templates/GUI_TEMPLATE_CRYO_CPA
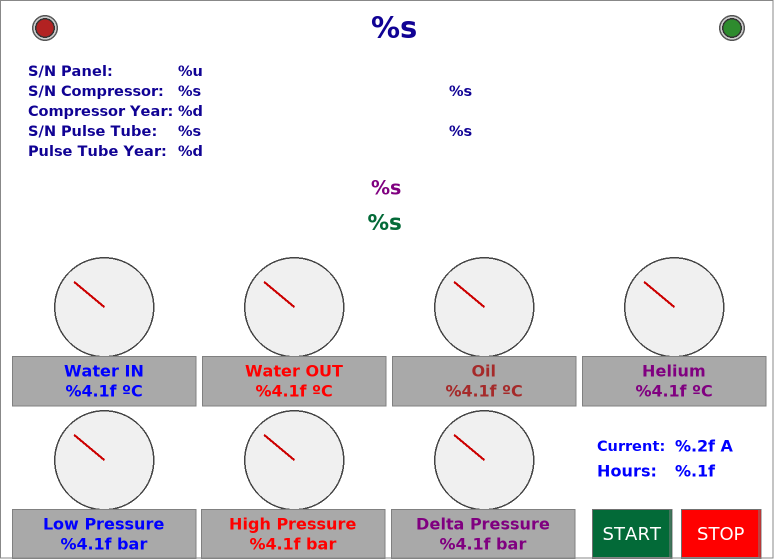
VISUALIZATION GUI_TEMPLATE_CRYO_CPA  // 774x559
VAR_IN_OUT
	m_Instance:	FB_CRYO_CPA;
END_VAR
    Rectangle (80,10 629x35), "%s", text variable: m_Instance.stat.sModelNumber
    Rectangle (10,207 750x30), "%s", text variable: m_Instance.stat.sError, invisible if: (m_Instance.stat.nStatusCode<>2)
    Meter180 (4,410 200x100), value: m_Instance.stat.lrLowPressure, style: Meter-Meter180-Gray, scale format: %.0f, scale 0..30
    Rectangle (12,509 184x50), "Low Pressure %4.1f bar", text variable: m_Instance.stat.lrLowPressure
    Meter180 (194,410 200x100), value: m_Instance.stat.lrHighPressure, style: Meter-Meter180-Gray, scale format: %.0f, scale 0..30
    Rectangle (201,509 184x50), "High Pressure %4.1f bar", text variable: m_Instance.stat.lrHighPressure
    Lamp1 (717,13 30x30), tooltip "If ON, compressor is running", variable: m_Instance.stat.bSystemOn, style: Lamp-Lamp1-Green
    Rectangle (10,208 750x30), "%s", text variable: m_Instance.stat.sAlarm, invisible if: (m_Instance.stat.nStatusCode<>1)
    Rectangle (231,206 308x33), "%s", text variable: m_Instance.stat.sStatusOK, invisible if: (m_Instance.stat.nStatusCode<>0 or m_Instance.stat.nOperatingState <>3)
    Meter180 (4,257 200x100), value: m_Instance.stat.lrCoolantInTemp, style: Meter-Meter180-Gray, scale format: %.0f, scale 0..60
    Rectangle (12,356 184x50), "Water IN %4.1f ºC", text variable: m_Instance.stat.lrCoolantInTemp
    Meter180 (194,257 200x100), value: m_Instance.stat.lrCoolantOutTemp, style: Meter-Meter180-Gray, scale format: %.0f, scale 0..60
    Rectangle (202,356 184x50), "Water OUT %4.1f ºC", text variable: m_Instance.stat.lrCoolantOutTemp
    Meter180 (384,257 200x100), value: m_Instance.stat.lrOilTemp, style: Meter-Meter180-Gray, scale format: %.0f, scale 0..60
    Rectangle (392,356 184x50), "Oil %4.1f ºC", text variable: m_Instance.stat.lrOilTemp
    Meter180 (574,257 200x100), value: m_Instance.stat.lrHeliumTemp, style: Meter-Meter180-Gray, scale format: %.0f, scale 0..100
    Rectangle (582,356 184x50), "Helium %4.1f ºC", text variable: m_Instance.stat.lrHeliumTemp
    Rectangle (672,431 95x30), "%.2f A", text variable: m_Instance.stat.lrMotorCurrent
    Rectangle (672,456 95x30), "%.1f", text variable: m_Instance.stat.lrHoursOfOperation
    Rectangle (140,173 493x30), "%s", tooltip "Operational State", text variable: m_Instance.stat.sOperatingState
    Rectangle (175,60 231x22), "%u", text variable: m_Instance.stat.nPanelSerialNumber
    Rectangle (175,80 270x22), "%s", text variable: m_Instance.in_sSN_Compressor
    Rectangle (175,120 270x22), "%s", text variable: m_Instance.in_sSN_PulseTube
    Label (25,60 145x22), "S/N Panel:"
    Label (25,80 145x22), "S/N Compressor:"
    Label (25,120 145x22), "S/N Pulse Tube:"
    Rectangle (594,431 75x30), "Current:"
    Rectangle (594,456 75x30), "Hours:"
    Meter180 (384,410 200x100), value: m_Instance.stat.lrDeltaPressureAverage, style: Meter-Meter180-Gray, scale format: %.0f, scale 0..30
    Rectangle (391,509 184x50), "Delta Pressure %4.1f bar", text variable: m_Instance.stat.lrDeltaPressureAverage
    Label (25,140 145x22), "Pulse Tube Year:"
    Rectangle (175,140 90x22), "%d", text variable: m_Instance.in_nYear_PulseTube
    Label (25,100 145x22), "Compressor Year:"
    Rectangle (175,100 90x22), "%d", text variable: m_Instance.in_nYear_Compressor
    Rectangle (446,80 270x22), "%s", text variable: m_Instance.stat.sServiceDue_Compressor, invisible if: m_Instance.stat.bServiceDue_Compressor=FALSE
        p55702900: m_Instance.stat.wColour_Compressor
    Rectangle (446,120 270x22), "%s", text variable: m_Instance.stat.sServiceDue_PulseTube, invisible if: m_Instance.stat.bServiceDue_PulseTube=FALSE
        p55702900: m_Instance.stat.wColour_PulseTube
    Button (592,509 80x50), "START", input disabled if: m_Instance.stat.bSystemOn
        OnMouseClick: execute { m_Instance.ctrl.nDevCommand := E_CRYO_CPA_CMDS.START; m_Instance.ctrl.bExecute := TRUE; }
    Button (681,509 80x50), "STOP", input disabled if: NOT m_Instance.stat.bSystemOn
        OnMouseClick: execute { m_Instance.ctrl.nDevCommand := E_CRYO_CPA_CMDS.STOP; m_Instance.ctrl.bExecute := TRUE; }
    Lamp1 (30,13 30x30), tooltip "If ON, compressor is simulated", variable: m_Instance.stat.bSimulation, invisible if: m_Instance.stat.bSimulation=false, style: Lamp-Lamp1-Red
END_VISUALIZATION

// VISUs/Templates/GUI_TEMPLATE_CRYO_EVAC_BASE
